(* Logix 5000 project; controller P4 vendor 1 type 14 code 92 rev 20.55; software revision 20.01 *)

TASK MainTask (continuous, watchdog 500 ms) : MainProgram

MODULES
   Local : vendor 1 type 14 code 92 (ICP 0, rev 20.55)
      P4_EN2T_PCN : 1756-EN2T (ICP 1, Ethernet 192.168.1.40, rev 10.1)
         P5 : 1756-EN2T (Ethernet 192.168.1.50, rev 10.1, Output RPI 10 ms)
            P5_CONTROLLER : vendor 1 type 14 code 92 (ICP 0, rev 20.1)
         P3 : 1756-EN2T (Ethernet 192.168.1.30, rev 10.7, Output RPI 10 ms)
            P3_CONTROLLER : vendor 1 type 14 code 92 (ICP 0, rev 20.55)
      P4_EN2TR_RIO : vendor 1 type 12 code 200 (ICP 2, Ethernet 192.168.0.40, rev 10.1)
         RIO4 : 1794-AENTR (Ethernet 192.168.0.42, rev 1.1, Output RPI 20 ms)
            RIO4_DI : 1794-IB32 (Flex 0, rev 1.1, Input RPI 20 ms)
            RIO4_DO : vendor 1 type 7 code 35 (Flex 1, rev 1.1)
            RIO4_AI : 1794-IE12 (Flex 2, rev 1.1, Output RPI 78 ms)
         WRIO4 : vendor 309 type 12 code 1000 (Ethernet 192.168.0.45, rev 3.1, Output RPI 20 ms)
            WRIO3_AI : 1734-IE4C (PointIO 1, rev 3.1, Input RPI 80 ms)
END_MODULES

TYPE AIN_UDT :
STRUCT
   Pv : REAL;
   Heu : REAL;
   Leu : REAL;
   SAHH : REAL;
   SAH : REAL;
   SAL : REAL;
   SALL : REAL;
   AHH : BOOL;
   AH : BOOL;
   AL : BOOL;
   ALL : BOOL;
   Wifi_Enb : BOOL;
   Hty : BOOL;
   Sim : BOOL;
   Sim_PV : REAL;
END_STRUCT
END_TYPE

TYPE AUTOINP_UDT :
STRUCT
   ON : BOOL;
END_STRUCT
END_TYPE

TYPE ControllerLEDStatus :
STRUCT
   Off : BOOL;
   SolidGreen : BOOL;
   FlashingGreen : BOOL;
   SolidYellow : BOOL;
   FlashingYellow : BOOL;
   FlashingRed : BOOL;
   SolidRed : BOOL;
END_STRUCT
END_TYPE

TYPE DOSING_SETPOINT_UDT :
STRUCT
   High_Setpoint : REAL;
   Low_Setpoint : REAL;
END_STRUCT
END_TYPE

TYPE Duty2_UDT :
STRUCT
   Selection : INT;
   Pump_Running : BOOL;
   Selected_Pmp_Not_Avl : BOOL;
   Both_Pmp_Not_Avl : BOOL;
END_STRUCT
END_TYPE

TYPE FaultRecord :
STRUCT
   timelow : DINT;
   timehigh : DINT;
   type : INT;
   code : INT;
   info : DINT[8];
END_STRUCT
END_TYPE

TYPE FIT_UDT :
STRUCT
   Pv : REAL;
   Heu : REAL;
   Leu : REAL;
   SAHH : REAL;
   SAH : REAL;
   SAL : REAL;
   SALL : REAL;
   Totaliser : REAL;
   AHH : BOOL;
   AH : BOOL;
   AL : BOOL;
   ALL : BOOL;
   Sim : BOOL;
   Sim_PV : REAL;
   Wifi_Enb : BOOL;
   Rst_Totaliser : BOOL;
   Hty : BOOL;
END_STRUCT
END_TYPE

TYPE Logix_Status_FP :
STRUCT
   ClearMinorFaults : DINT;
   Sts_MinorFaultEvents : DINT;
   Sts_MinorFaultBits : DINT;
   Sts_Redundant : DINT;
   Set_FaceplateAnimation : DINT;
   Val_ProductCode : DINT;
   MemoryTemp : INT[29];
   Val_raw_data : INT;
   Sts_IO_LED_raw : INT;
   Sts_ProductCode : INT;
   Val_Force_data_raw : INT;
   MemoryRequestData : SINT[12];
   Sts_Force_Installed : BOOL;
   Sts_Force_Enabled : BOOL;
   Sts_Faulted : BOOL;
   Sts_Run : BOOL;
   Sts_Program : BOOL;
   Sts_Minor_fault : BOOL;
   Sts_Major_fault : BOOL;
   Sts_KS_in_run : BOOL;
   Sts_KS_in_program : BOOL;
   Sts_KS_in_remote : BOOL;
   Sts_Changingmodes : BOOL;
   Sts_Test : BOOL;
   Sts_Ladder_Working : BOOL;
   Cmd_ClearFaultRecord : BOOL;
   Set_Controller_Description : STRING;
   UpdateDelayTimer : TIMER;
   Val_MajorFault : FaultRecord;
   Val_MFS : FaultRecord;
   Sts_IO_LED : ControllerLEDStatus;
   Sts_Battery_LED : ControllerLEDStatus;
   MemoryData : Memory_Data;
   TEST : DINT;
END_STRUCT
END_TYPE

TYPE Memory_Data :
STRUCT
   Free_Mem_IO : DINT;
   Free_Mem_DT : DINT;
   Free_Memory : DINT;
   Total_Mem_IO : DINT;
   Total_Mem_DT : DINT;
   Total_Memory : DINT;
   Biggest_IO_Mem_Size_Ava : DINT;
   Biggest_DT_Mem_Size_Ava : DINT;
END_STRUCT
END_TYPE

TYPE MV_UDT :
STRUCT
   Cmd : INT;
   Status : INT;
   Reset : BOOL;
   Auto : BOOL;
   FTO : BOOL;
   FTC : BOOL;
   Avl : BOOL;
END_STRUCT
END_TYPE

TYPE PLANT_AUTO_UDT :
STRUCT
   ON : BOOL;
   OFF : BOOL;
END_STRUCT
END_TYPE

TYPE PLANT_UDT :
STRUCT
   START : BOOL;
   STOP : BOOL;
END_STRUCT
END_TYPE

TYPE PMP_UDT :
STRUCT
   Cmd : INT;
   Status : INT;
   RunMin : REAL;
   Total_RunMin : REAL;
   RunHr : REAL;
   Total_RunHr : REAL;
   Remote : BOOL;
   Auto : BOOL;
   Fault : BOOL;
   Avl : BOOL;
   Permissive : DINT;
   Shutdown : DINT;
   SD : DINT;
   Reset : BOOL;
   Reset_RunHr : BOOL;
   FTR : BOOL;
   FTS : BOOL;
END_STRUCT
END_TYPE

TYPE PRECONDITION_UDT :
STRUCT
   PERMISSIVE1 : BOOL;
   PERMISSIVE2 : BOOL;
   PERMISSIVE3 : BOOL;
   PERMISSIVE4 : BOOL;
   PERMISSIVE5 : BOOL;
   SHUTDOWN1 : BOOL;
   SHUTDOWN2 : BOOL;
   SHUTDOWN3 : BOOL;
   SHUTDOWN4 : BOOL;
   SHUTDOWN5 : BOOL;
END_STRUCT
END_TYPE

TYPE RED_STAT :
STRUCT
   Redundancy_status_of_the_controller : INT;
   Redundancy_state_of_the_partner : INT;
END_STRUCT
END_TYPE

TYPE SWITCH_UDT :
STRUCT
   Alarm : BOOL;
   Delay : DINT;
END_STRUCT
END_TYPE

TYPE UV_UDT :
STRUCT
   Cmd : INT;
   Status : INT;
   RunMin : REAL;
   Total_RunMin : REAL;
   RunHr : REAL;
   Total_RunHr : REAL;
   Remote : BOOL;
   Auto : BOOL;
   Fault : BOOL;
   Avl : BOOL;
   Permissive : DINT;
   Shutdown : DINT;
   SD : DINT;
   Reset : BOOL;
   Reset_RunHr : BOOL;
   FTR : BOOL;
   FTS : BOOL;
END_STRUCT
END_TYPE

TYPE WIFI_UDT :
STRUCT
   PLC_WIFI : BOOL;
   RIO_WIFI : BOOL;
END_STRUCT
END_TYPE

ADD_ON_INSTRUCTION AIN_FBD   (* revision 1.0 *)
VAR_INPUT
   WRIO_Enb : BOOL; {visible}
   Raw_RIO : INT; {visible}
   Raw_WRIO : INT; {visible}
   L_Raw_RIO : INT; {visible}
   H_Raw_RIO : INT; {visible}
   L_Raw_WRIO : INT; {visible}
   H_Raw_WRIO : INT; {visible}
   HEU : INT; {visible}
   LEU : INT; {visible}
END_VAR
VAR_OUTPUT
   Hty : BOOL; {visible}
   Wifi_Enb : BOOL; {access Read Only, visible}
   AHH : BOOL; {visible}
   AH : BOOL; {access Read Only, visible}
   AL : BOOL; {access Read Only, visible}
   ALL : BOOL; {visible}
END_VAR
VAR_INPUT
   SAHH : REAL; {visible}
   SAH : REAL; {visible}
   SAL : REAL; {visible}
   SALL : REAL; {visible}
   Simulation : BOOL; {visible}
   RIO_Hty : BOOL; {visible}
   WRIO_Hty : BOOL; {visible}
END_VAR
VAR_IN_OUT
   Pv : REAL; {required}
   Sim_PV : REAL; {required}
   HMI : AIN_UDT; {required}
END_VAR
VAR
   SCALE : SCALE; {access None}
   ALM : ALARM; {access None}
   _Raw : INT; {access None}
   _L_Raw : INT; {access None}
   _H_Raw : INT; {access None}
   _Inst_Hty : BOOL; {access None}
END_VAR

ROUTINE Logic   (* structured text *)
   (*RIO and Wireless RIO Selection*)
   
   IF WRIO_Enb THEN
   	Wifi_Enb	:= 1;
   	_Raw		:= Raw_WRIO;
   	_H_Raw		:= H_Raw_WRIO;
   	_L_Raw		:= L_Raw_WRIO;
   	_Inst_Hty 	:= WRIO_Hty;
   ELSE
   	Wifi_Enb	:= 0;
   	_Raw		:= Raw_RIO;
   	_H_Raw		:= H_Raw_RIO;
   	_L_Raw		:= L_Raw_RIO;
   	_Inst_Hty 	:= RIO_Hty;
   END_IF;
   
   (*Calculation for PV*)
   IF Simulation THEN
   	Pv	:=Sim_PV;
   ELSE
   	SCALE.In		:=_Raw;
   	SCALE.InRawMax	:=_H_Raw;
   	SCALE.InRawMin	:=_L_Raw;
   	SCALE.InEUMax	:=HEU;
   	SCALE.InEUMin	:=LEU;
   	SCL(SCALE);
   
   	IF SCALE.Out<0 THEN
   		Pv	:= 0.0;
   	ELSE
   		Pv	:=SCALE.Out;
   	END_IF;
   
   	Sim_PV	:=Pv;
   
   END_IF;
   
   (*Alarms*)
   ALM.In			:=Pv;
   ALM.HHLimit		:=SAHH;
   ALM.HLimit		:=SAH;
   ALM.LLimit		:=SAL;
   ALM.LLLimit		:=SALL;
   ALM(ALM);
   
   AHH				:=ALM.HHAlarm;
   AH				:=ALM.HAlarm;
   AL				:=ALM.LAlarm;
   ALL				:=ALM.LLAlarm;
   
   Hty:= _Inst_Hty AND (_Raw > _L_Raw) AND (_Raw < _H_Raw)  ;
   
   
   
   
   
   
END_ROUTINE
END_ADD_ON_INSTRUCTION

ADD_ON_INSTRUCTION Duty2_FBD   (* revision 1.0 *)
VAR_INPUT
   AutoInp : BOOL; {visible}
   Selection : INT; {visible}
END_VAR
VAR_OUTPUT
   Start_Pmp1 : BOOL; {visible}
   Start_Pmp2 : BOOL; {visible}
END_VAR
VAR_IN_OUT
   PMP1 : PMP_UDT; {required}
   PMP2 : PMP_UDT; {required}
   HMI : Duty2_UDT; {required}
END_VAR

ROUTINE Logic   (* structured text *)
   IF PMP1.Status=2 OR PMP2.Status=2 THEN
   	HMI.Pump_Running := 1;
   ELSE
   	HMI.Pump_Running := 0;
   END_IF;
   
   HMI.Both_Pmp_Not_Avl		:= NOT PMP1.Avl AND NOT PMP2.Avl;
   
   IF AutoInp THEN
   	CASE Selection OF
   		(*PUMP 1 *)
   		1:
   			IF PMP1.Avl THEN
   				Start_Pmp1					:=1;
   				Start_Pmp2					:=0;
   				HMI.Selected_Pmp_Not_Avl	:=0;
   			ELSIF NOT PMP1.Avl AND PMP2.Avl THEN
   				Start_Pmp1					:=0;
   				Start_Pmp2					:=1;
   				HMI.Selected_Pmp_Not_Avl	:=1;
   			ELSIF NOT PMP1.Avl AND NOT PMP2.Avl	THEN
   				Start_Pmp1					:=0;
   				Start_Pmp2					:=0;
   			ELSE
   				HMI.Selected_Pmp_Not_Avl	:=0;
   			END_IF;
   
   		(*PUMP 2 *)
   		2:
   			IF PMP2.Avl THEN
   				Start_Pmp1					:=0;
   				Start_Pmp2					:=1;
   				HMI.Selected_Pmp_Not_Avl	:=0;
   			ELSIF NOT PMP2.Avl AND PMP1.Avl THEN
   				Start_Pmp1					:=1;
   				Start_Pmp2					:=0;
   				HMI.Selected_Pmp_Not_Avl	:=1;
   			ELSIF NOT PMP1.Avl AND NOT PMP2.Avl	THEN
   				Start_Pmp1					:=0;
   				Start_Pmp2					:=0;
   			ELSE
   				HMI.Selected_Pmp_Not_Avl	:=0;
   			END_IF;
   	END_CASE;
   ELSE
   	Start_Pmp1					:=0;
   	Start_Pmp2					:=0;
   END_IF;
   
   
END_ROUTINE
END_ADD_ON_INSTRUCTION

ADD_ON_INSTRUCTION FIT_FBD   (* revision 1.0 *)
VAR_INPUT
   WRIO_Enb : BOOL; {visible}
   Raw_RIO : INT; {visible}
   Raw_WRIO : INT; {visible}
   L_Raw_RIO : INT; {visible}
   H_Raw_RIO : INT; {visible}
   L_Raw_WRIO : INT; {visible}
   H_Raw_WRIO : INT; {visible}
   HEU : REAL; {visible}
   LEU : REAL; {visible}
END_VAR
VAR_OUTPUT
   Hty : BOOL; {visible}
   Wifi_Enb : BOOL; {visible}
   AHH : BOOL; {visible}
   AH : BOOL; {access Read Only, visible}
   AL : BOOL; {access Read Only, visible}
   ALL : BOOL; {visible}
END_VAR
VAR_INPUT
   SAHH : REAL; {visible}
   SAH : REAL; {visible}
   SAL : REAL; {visible}
   SALL : REAL; {visible}
   Simulation : BOOL; {visible}
   RIO_Hty : BOOL; {visible}
   WRIO_Hty : BOOL; {visible}
   Totaliser_Enb : BOOL; {visible}
   Rst_Totaliser : BOOL; {visible}
END_VAR
VAR_IN_OUT
   Totaliser : REAL; {required}
   Pv : REAL; {required}
   Sim_Pv : REAL; {required}
   HMI : FIT_UDT; {required}
END_VAR
VAR
   SCALE : SCALE; {access None}
   ALM : ALARM; {access None}
   TON : FBD_TIMER; {access None}
   _SEC_P : BOOL; {access None}
   _Inst_Hty : BOOL; {access None}
   _L_Raw : INT; {access None}
   _H_Raw : INT; {access None}
   _Raw : INT; {access None}
   R_TRIG : FBD_ONESHOT; {access None}
END_VAR

ROUTINE Logic   (* structured text *)
   (*RIO and Wireless RIO Selection*)
   
   IF WRIO_Enb THEN
   	Wifi_Enb	:= 1;
   	_Raw		:= Raw_WRIO;
   	_H_Raw		:= H_Raw_WRIO;
   	_L_Raw		:= L_Raw_WRIO;
   	_Inst_Hty 	:= WRIO_Hty;
   ELSE
   	Wifi_Enb	:= 0;
   	_Raw		:= Raw_RIO;
   	_H_Raw		:= H_Raw_RIO;
   	_L_Raw		:= L_Raw_RIO;
   	_Inst_Hty 	:= RIO_Hty;
   END_IF;
   
   (*Calculation for PV*)
   IF Simulation THEN
   	Pv	:= Sim_Pv   ;
   ELSE
   	SCALE.In		:=_Raw;
   	SCALE.InRawMax	:=_H_Raw;
   	SCALE.InRawMin	:=_L_Raw;
   	SCALE.InEUMax	:=HEU;
   	SCALE.InEUMin	:=LEU;
   	SCL(SCALE);
   	IF SCALE.Out>0 THEN
   		Pv	:=SCALE.Out;
   	ELSIF SCALE.Out<=0 THEN
   		Pv	:=0.0;
   	END_IF;
   
   	Sim_Pv	:=Pv;
   END_IF;
   
   (*Alarms*)
   ALM.In			:=Pv;
   ALM.HHLimit		:=SAHH;
   ALM.HLimit		:=SAH;
   ALM.LLimit		:=SAL;
   ALM.LLLimit		:=SALL;
   ALM(ALM);
   
   AHH				:=ALM.HHAlarm;
   AH				:=ALM.HAlarm;
   AL				:=ALM.LAlarm;
   ALL				:=ALM.LLAlarm;
   
   (*SECOND PULSE*)
   TON.PRE	:=1000;
   TON.TimerEnable	:=1;
   TONR(TON );
   R_TRIG.InputBit :=TON.DN ;
   OSRI( R_TRIG);
   _SEC_P  := R_TRIG.OutputBit;
   TON.Reset := _SEC_P;
   
   IF Totaliser_Enb THEN
   	IF _SEC_P THEN
   		HMI.Totaliser := HMI.Totaliser +  (ABS(Pv) / 3600 );
   	END_IF;
   END_IF;
   
   IF  Rst_Totaliser   THEN
   	HMI.Totaliser	:=0;
   END_IF;
   
   Hty:= _Inst_Hty AND (_Raw > _L_Raw) AND (_Raw < _H_Raw)  ;
   
   
   
   
   
   
END_ROUTINE
END_ADD_ON_INSTRUCTION

ADD_ON_INSTRUCTION MV_FBD   (* revision 1.0 *)
VAR_INPUT
   Auto : BOOL; {visible}
END_VAR
VAR_OUTPUT
   Cmd_Open : BOOL; {visible}
   Cmd_Close : BOOL; {visible}
   FTO : BOOL; {visible}
   FTC : BOOL; {access Read Only, visible}
END_VAR
VAR_INPUT
   AutoInp : BOOL; {visible}
   ZSO : BOOL; {visible}
   Open_TM : DINT; {visible}
   ZSC : BOOL; {visible}
   Close_TM : DINT; {visible}
END_VAR
VAR_IN_OUT
   Cmd : INT; {required}
   HMI : MV_UDT; {required}
END_VAR
VAR
   TON_Open_TM : FBD_TIMER; {access None}
   TON_Close_TM : FBD_TIMER; {access None}
END_VAR

ROUTINE Logic   (* structured text *)
   (*Fail to Close*)
   TON_Close_TM.PRE 			:= 	Close_TM*1000;
   TON_Close_TM.TimerEnable 	:=  Cmd_Close;
   TONR(TON_Close_TM);
   
   (*Fail to Open*)
   TON_Open_TM.PRE 			:= 	Open_TM*1000;
   TON_Open_TM.TimerEnable 	:= 	Cmd_Open;
   TONR(TON_Open_TM);
   
   IF ZSC THEN
   	HMI.Status	:=1;
   ELSIF ZSO THEN
   	HMI.Status	:=2;
   ELSE
   	HMI.Status	:=0;
   END_IF;
   
   HMI.Avl:= Auto AND NOT FTC AND NOT FTO;
   
   IF HMI.Reset THEN
   	(*IF NOT TON_Close_TM.DN AND ZSC THEN*)
   			FTC		:= 0;
   	(*END_IF;*)
   	(*IF NOT TON_Open_TM.DN AND ZSO THEN*)
   			FTO		:= 0;
   	(*END_IF;*)
   END_IF;
   
   IF  NOT Auto THEN
   	CASE HMI.Cmd OF
   		1:	(*CLOSE*)
   			Cmd_Close	:= 1;
   			Cmd_Open	:= 0;
   			IF TON_Close_TM.DN AND (NOT ZSC) THEN
   				FTC		:= 1;
   				FTO		:= 0;
   			END_IF;
   		2:	(*OPEN*)
   			IF FTO OR FTC    THEN
   				HMI.Cmd := 1;
   			END_IF;
   
   			IF NOT FTC AND NOT FTO THEN
   				Cmd_Close	:= 0;
   				Cmd_Open	:= 1;
   			END_IF;
   
   			IF TON_Open_TM.DN AND (NOT ZSO) THEN
   				FTC		:= 0;
   				FTO		:= 1;
   				HMI.Cmd := 1;
   			END_IF;
   	END_CASE;
   ELSE
   	(*Maintain Last status when switching from Auto to Manual*)
   	IF ZSO THEN
   		Cmd	:= 2;
   	END_IF;
   	IF ZSC THEN
   		Cmd	:= 1;
   	END_IF;
   
   	IF  AutoInp AND (NOT FTC AND NOT FTO) THEN
   		Cmd_Close	:= 0;
   		Cmd_Open	:= 1;
   		IF TON_Open_TM.DN AND (NOT ZSO) THEN
   			FTC		:= 0;
   			FTO		:= 1;
   		END_IF;
   	ELSE
   		Cmd_Close	:= 1;
   		Cmd_Open	:= 0;
   		IF TON_Close_TM.DN AND (NOT ZSC) THEN
   			FTC		:= 1;
   			FTO		:= 0;
   		END_IF;
   	END_IF;
   END_IF;
   
   
END_ROUTINE
END_ADD_ON_INSTRUCTION

ADD_ON_INSTRUCTION PMP_FBD   (* revision 1.0 *)
VAR_OUTPUT
   Cmd_Start : BOOL; {visible}
   Avl : BOOL; {visible}
   Fault : BOOL; {visible}
   FT_Stop : BOOL; {visible}
   FT_Start : BOOL; {visible}
   RunHr : REAL; {visible}
   Total_RunHr : REAL; {visible}
   SD : DINT; {access Read Only, visible}
END_VAR
VAR_INPUT
   Auto : BOOL; {visible}
   AutoInp : BOOL; {visible}
   Remote : BOOL; {visible}
   Run : BOOL; {visible}
   Trip : BOOL; {visible}
   Start_TM : DINT; {visible}
   Stop_TM : DINT; {visible}
   Rst : BOOL; {visible}
   Rst_RunHr : BOOL; {visible}
   Permissive : DINT; {visible}
   Shutdown : DINT; {visible}
END_VAR
VAR_IN_OUT
   RunMin : REAL; {required}
   Total_RunMin : REAL; {required}
   Cmd : INT; {required}
   HMI : PMP_UDT; {required}
END_VAR
VAR
   TON_Start_TM : FBD_TIMER; {access None}
   TON_Stop_TM : FBD_TIMER; {access None}
   _Min_P : BOOL; {access None}
   TON_Min : FBD_TIMER; {access None}
   R_TRIG_SEC : FBD_ONESHOT; {access None}
END_VAR

ROUTINE Logic   (* structured text *)
   (*Fail to Start*)
   TON_Start_TM.PRE 			:= 	Start_TM*1000;
   TON_Start_TM.TimerEnable 	:=  Cmd_Start;
   TONR(TON_Start_TM);
   
   (*Fail to Stop*)
   TON_Stop_TM.PRE 			:= 	Stop_TM*1000;
   TON_Stop_TM.TimerEnable 	:=  NOT Cmd_Start;
   TONR(TON_Stop_TM);
   
   IF (NOT Run) THEN
   	HMI.Status	:=1;
   ELSE
   	HMI.Status	:=2;
   END_IF;
   
   IF Fault THEN
   	HMI.Fault:= 1;
   ELSE
   	HMI.Fault:= 0;
   END_IF;
   
   IF HMI.Reset THEN
   	IF NOT TON_Stop_TM.DN THEN
   			FT_Stop		:= 0;
   	END_IF;
   	IF NOT TON_Start_TM.DN THEN
   			FT_Start	:= 0;
   	END_IF;
   
   	SD :=0;
   
   END_IF;
   
   Fault		:=Trip OR SD<>0;
   HMI.Remote	:=Remote;
   Avl:= Auto AND Remote AND NOT Fault AND NOT FT_Start AND NOT FT_Stop AND SD=0 ;
   
   IF Remote THEN
   	IF  NOT Auto THEN
   		CASE HMI.Cmd OF
   			1:	(*Stop*)
   				Cmd_Start	:=0;
   				IF TON_Stop_TM.DN AND Run THEN
   					FT_Start	:= 0;
   					FT_Stop		:= 1;
   				END_IF;
   			2:	(*OPEN*)
   				IF NOT Fault AND NOT FT_Start AND NOT FT_Stop AND (Permissive=-1) AND HMI.SD=0 THEN
   					Cmd_Start	:= 1;
   				ELSIF Cmd_Start AND (HMI.SD<>0) OR Fault THEN
   					SD				:= HMI.SD;
   					Cmd_Start		:= 0;
   					HMI.Cmd 		:= 1;
   				ELSIF (Permissive<>-1) THEN
   					HMI.Cmd 		:= 1;
   				END_IF;
   
   				IF TON_Start_TM.DN AND NOT Run THEN
   					FT_Start	:= 1;
   					FT_Stop		:= 0;
   					Cmd_Start	:= 0;
   					HMI.Cmd 	:= 1;
   				END_IF;
   		END_CASE;
   	ELSE
   		IF Run THEN
   			Cmd	:= 2;
   		END_IF;
   		IF (NOT Run) OR Fault OR FT_Start OR FT_Stop THEN
   			Cmd	:= 1;
   		END_IF;
   
   		IF  AutoInp  THEN
   			IF NOT Fault AND NOT FT_Start AND NOT FT_Stop AND (Permissive=-1) AND HMI.SD=0  THEN
   				Cmd_Start	:=1;
   			ELSIF Cmd_Start OR (HMI.SD<>0) OR Fault THEN
   				SD			:= HMI.SD;
   				Cmd_Start	:=0;
   			END_IF;
   
   			IF TON_Start_TM.DN AND NOT Run THEN
   				FT_Start	:= 1;
   				FT_Stop		:= 0;
   				Cmd_Start	:= 0;
   				HMI.Cmd 	:= 1;
   			END_IF;
   		ELSE
   			Cmd_Start	:=0;
   			IF TON_Stop_TM.DN AND Run THEN
   				FT_Start	:= 0;
   				FT_Stop		:= 1;
   
   			END_IF;
   		END_IF;
   	END_IF;
   
   ELSE (*Local*)
   	Cmd_Start	:=0;
   	Cmd	:= 1;
   
   	FT_Start	:= 0;
   	FT_Stop		:= 0;
   
   
   
   
   	(*	IF Run THEN
   			Cmd	:= 2;
   		END_IF;
   		IF (NOT Run) OR Fault OR FT_Start OR FT_Stop THEN
   			Cmd	:= 1;
   		END_IF;
   		*)
   END_IF;
   
   (*1 MIN PULSE*)
   TON_Min.PRE	:=60000;
   TON_Min.TimerEnable	:=1;
   TONR(TON_Min );
   R_TRIG_SEC.InputBit :=TON_Min.DN ;
   OSRI( R_TRIG_SEC);
   _Min_P  := R_TRIG_SEC.OutputBit;
   TON_Min.Reset 	:= _Min_P;
   
   IF Run THEN
   	IF _Min_P THEN
   		RunMin 			:=RunMin + 1.0;
   		Total_RunMin	:=Total_RunMin + 1.0;
   	END_IF;
   END_IF;
   
   RunHr 				:=RunMin/60.0;
   Total_RunHr			:=Total_RunMin/60.0;
   
   IF  Rst_RunHr THEN
   	RunMin	:=0;
   END_IF;
   
   
   
END_ROUTINE
END_ADD_ON_INSTRUCTION

ADD_ON_INSTRUCTION SWITCH_FBD   (* revision 1.0 *)
VAR_INPUT
   Alarm : BOOL; {visible}
   Delay : DINT; {required}
END_VAR
VAR_OUTPUT
   Status : BOOL; {access None, required}
END_VAR
VAR_IN_OUT
   HMI : SWITCH_UDT; {required}
END_VAR
VAR
   TON_Delay_Sec : FBD_TIMER; {access None}
END_VAR

ROUTINE Logic   (* structured text *)
   (*Delay for Alarm*)
   TON_Delay_Sec.PRE 			:= 	Delay*1000;
   TON_Delay_Sec.TimerEnable 	:=  Alarm;
   TONR(TON_Delay_Sec);
   
   Status := TON_Delay_Sec.DN ;
END_ROUTINE
END_ADD_ON_INSTRUCTION

ADD_ON_INSTRUCTION UV_FBD   (* revision 1.0 *)
VAR_OUTPUT
   Cmd_Start : BOOL; {visible}
   Avl : BOOL; {visible}
   Fault : BOOL; {visible}
   FT_Stop : BOOL; {visible}
   FT_Start : BOOL; {visible}
   RunHr : REAL; {visible}
   Total_RunHr : REAL; {visible}
   SD : DINT; {visible}
END_VAR
VAR_INPUT
   Auto : BOOL; {visible}
   AutoInp : BOOL; {visible}
   Remote : BOOL; {visible}
   Run : BOOL; {visible}
   Trip : BOOL; {visible}
   Start_TM : DINT; {visible}
   Stop_TM : DINT; {visible}
   Rst : BOOL; {visible}
   Rst_RunHr : BOOL; {visible}
   Permissive : DINT; {visible}
   Shutdown : DINT; {visible}
END_VAR
VAR_IN_OUT
   RunMin : REAL; {required}
   Total_RunMin : REAL; {required}
   Cmd : INT; {required}
   HMI : UV_UDT; {required}
END_VAR
VAR
   TON_Start_TM : FBD_TIMER; {access None}
   TON_Stop_TM : FBD_TIMER; {access None}
   _Min_P : BOOL; {access None}
   TON_Min : FBD_TIMER; {access None}
   R_TRIG_SEC : FBD_ONESHOT; {access None}
END_VAR

ROUTINE Logic   (* structured text *)
   (*Fail to Start*)
   TON_Start_TM.PRE 			:= 	Start_TM*1000;
   TON_Start_TM.TimerEnable 	:=  Cmd_Start;
   TONR(TON_Start_TM);
   
   (*Fail to Stop*)
   TON_Stop_TM.PRE 			:= 	Stop_TM*1000;
   TON_Stop_TM.TimerEnable 	:=  NOT Cmd_Start;
   TONR(TON_Stop_TM);
   
   IF (NOT Run) THEN
   	HMI.Status	:=1;
   ELSE
   	HMI.Status	:=2;
   END_IF;
   
   IF Fault THEN
   	HMI.Fault:= 1;
   ELSE
   	HMI.Fault:= 0;
   END_IF;
   
   IF HMI.Reset THEN
   	IF NOT TON_Stop_TM.DN THEN
   			FT_Stop		:= 0;
   	END_IF;
   	IF NOT TON_Start_TM.DN THEN
   			FT_Start	:= 0;
   	END_IF;
   
   	SD :=0;
   
   END_IF;
   
   Fault		:=Trip;
   HMI.Remote	:=Remote;
   Avl:= Auto AND Remote AND NOT Fault AND NOT FT_Start AND NOT FT_Stop AND SD=0 ;
   
   IF Remote THEN
   	IF  NOT Auto THEN
   		CASE HMI.Cmd OF
   			1:	(*Stop*)
   				Cmd_Start	:=0;
   				IF TON_Stop_TM.DN AND Run THEN
   					FT_Start	:= 0;
   					FT_Stop		:= 1;
   				END_IF;
   			2:	(*OPEN*)
   				IF NOT Fault AND NOT FT_Start AND NOT FT_Stop AND (Permissive=-1) AND HMI.SD=0 THEN
   					Cmd_Start	:= 1;
   				ELSIF Cmd_Start AND (HMI.SD<>0) OR Fault THEN
   					SD				:= HMI.SD;
   					Cmd_Start		:= 0;
   					HMI.Cmd 		:= 1;
   				END_IF;
   
   				IF TON_Start_TM.DN AND NOT Run THEN
   					FT_Start	:= 1;
   					FT_Stop		:= 0;
   					Cmd_Start	:= 0;
   					HMI.Cmd 	:= 1;
   				END_IF;
   		END_CASE;
   	ELSE
   		IF Run THEN
   			Cmd	:= 2;
   		END_IF;
   		IF (NOT Run) OR Fault OR FT_Start OR FT_Stop THEN
   			Cmd	:= 1;
   		END_IF;
   
   		IF  AutoInp  THEN
   			IF NOT Fault AND NOT FT_Start AND NOT FT_Stop AND (Permissive=-1) AND HMI.SD=0  THEN
   				Cmd_Start	:=1;
   			ELSIF Cmd_Start OR (HMI.SD<>0) OR Fault THEN
   				SD			:= HMI.SD;
   				Cmd_Start	:=0;
   			END_IF;
   
   			IF TON_Start_TM.DN AND NOT Run THEN
   				FT_Start	:= 1;
   				FT_Stop		:= 0;
   				Cmd_Start	:= 0;
   				HMI.Cmd 	:= 1;
   			END_IF;
   		ELSE
   			Cmd_Start	:=0;
   			IF TON_Stop_TM.DN AND Run THEN
   				FT_Start	:= 0;
   				FT_Stop		:= 1;
   
   			END_IF;
   		END_IF;
   	END_IF;
   
   ELSE (*Local*)
   	Cmd_Start	:=0;
   	Cmd	:= 1;
   
   	FT_Start	:= 0;
   	FT_Stop		:= 0;
   
   
   
   
   	(*	IF Run THEN
   			Cmd	:= 2;
   		END_IF;
   		IF (NOT Run) OR Fault OR FT_Start OR FT_Stop THEN
   			Cmd	:= 1;
   		END_IF;
   		*)
   END_IF;
   
   (*1 MIN PULSE*)
   TON_Min.PRE	:=60000;
   TON_Min.TimerEnable	:=1;
   TONR(TON_Min );
   R_TRIG_SEC.InputBit :=TON_Min.DN ;
   OSRI( R_TRIG_SEC);
   _Min_P  := R_TRIG_SEC.OutputBit;
   TON_Min.Reset 	:= _Min_P;
   
   IF Run THEN
   	IF _Min_P THEN
   		RunMin 			:=RunMin + 1.0;
   		Total_RunMin	:=Total_RunMin + 1.0;
   	END_IF;
   END_IF;
   
   RunHr 				:=RunMin/60.0;
   Total_RunHr			:=Total_RunMin/60.0;
   
   IF  Rst_RunHr THEN
   	RunMin	:=0;
   END_IF;
   
   
   
END_ROUTINE
END_ADD_ON_INSTRUCTION

VAR_GLOBAL   (* controller tags *)
   _FIT401_Tot_Enb : BOOL;
   _P401_AutoInp : BOOL;
   _P402_AutoInp : BOOL;
   _P403_AutoInp : BOOL;
   _P404_AutoInp : BOOL;
   _P_NAHSO3_ORP_DUTY_AutoInp : BOOL;
   _P_NAHSO3_ORP_DUTY_SR : DOMINANT_SET := (Reset := 1, OutNot := 1);
   _P_RO_FEED_DUTY_AutoInp : BOOL;
   _P_RO_FEED_DUTY_SR : DOMINANT_SET := (Set := 1, Out := 1);
   _P_UF_FEED_DUTY_AutoInp : BOOL := 1;
   _UV401_AutoInp : BOOL;
   _UV_SR : DOMINANT_SET := (Set := 1, Out := 1);
   AI_AIT_401_HRDNSS : INT := 35;
   AI_AIT_401_HRDNSS_HTY : BOOL := 1;
   AI_AIT_402_ORP : INT := 9619;
   AI_AIT_402_ORP_HTY : BOOL := 1;
   AI_FIT_401_FLOW : INT := -7;
   AI_FIT_401_FLOW_HTY : BOOL := 1;
   AI_LIT_401_LEVEL : INT := 20593;
   AI_LIT_401_LEVEL_HTY : BOOL := 1;
   AI_RIO4_SPARE_03 : INT := 9619;
   AI_RIO4_SPARE_03_HTY : BOOL := 1;
   AI_RIO4_SPARE_04 : INT := -7703;
   AI_RIO4_SPARE_04_HTY : BOOL := 1;
   AI_RIO4_SPARE_05 : INT := -7703;
   AI_RIO4_SPARE_05_HTY : BOOL := 1;
   AI_RIO4_SPARE_06 : INT := -7698;
   AI_RIO4_SPARE_06_HTY : BOOL := 1;
   AI_RIO4_SPARE_07 : INT := -7702;
   AI_RIO4_SPARE_07_HTY : BOOL := 1;
   AI_RIO4_SPARE_08 : INT := -7699;
   AI_RIO4_SPARE_08_HTY : BOOL := 1;
   AI_RIO4_SPARE_09 : INT := -7702;
   AI_RIO4_SPARE_09_HTY : BOOL := 1;
   AI_RIO4_SPARE_10 : INT := -7701;
   AI_RIO4_SPARE_10_HTY : BOOL := 1;
   AI_RIO4_SPARE_11 : INT := -7703;
   AI_RIO4_SPARE_11_HTY : BOOL := 1;
   AIT401_FB : AIN_FBD := (Raw_RIO := 35, Raw_WRIO := 3261, H_Raw_RIO := 31208, L_Raw_WRIO := 3277, H_Raw_WRIO := 16383, HEU := 150, Hty := 1, AL := 1, ALL := 1, SAHH := 100.0, SAH := 80.0, SAL := 20.0, SALL := 10.0, RIO_Hty := 1, WRIO_Hty := 1);
   AIT401_FB_01 : AIN_FBD;
   AIT402_FB : AIN_FBD := (Raw_RIO := 9619, Raw_WRIO := 8246, H_Raw_RIO := 31208, L_Raw_WRIO := 3277, H_Raw_WRIO := 16383, HEU := 800, Hty := 1, AL := 1, SAHH := 800.0, SAH := 275.0, SAL := 250.0, SALL := 200.0, RIO_Hty := 1);
   DI_DPSH_301_HIGH : BOOL;
   DI_LS_401_LOW : BOOL := 1;
   DI_P_401_AUTO : BOOL := 1;
   DI_P_401_FAULT : BOOL;
   DI_P_401_RUN : BOOL;
   DI_P_402_AUTO : BOOL := 1;
   DI_P_402_FAULT : BOOL;
   DI_P_402_RUN : BOOL;
   DI_P_403_AUTO : BOOL := 1;
   DI_P_403_FAULT : BOOL;
   DI_P_403_RUN : BOOL;
   DI_P_404_AUTO : BOOL := 1;
   DI_P_404_FAULT : BOOL;
   DI_P_404_RUN : BOOL;
   DI_RIO4_SPARE_10 : BOOL;
   DI_RIO4_SPARE_11 : BOOL;
   DI_RIO4_SPARE_12 : BOOL;
   DI_RIO4_SPARE_13 : BOOL;
   DI_RIO4_SPARE_14 : BOOL;
   DI_RIO4_SPARE_15 : BOOL;
   DI_RIO4_SPARE_16 : BOOL;
   DI_RIO4_SPARE_17 : BOOL;
   DI_RIO4_SPARE_18 : BOOL;
   DI_RIO4_SPARE_19 : BOOL;
   DI_RIO4_SPARE_20 : BOOL;
   DI_RIO4_SPARE_21 : BOOL;
   DI_RIO4_SPARE_22 : BOOL;
   DI_RIO4_SPARE_23 : BOOL;
   DI_RIO4_SPARE_24 : BOOL;
   DI_RIO4_SPARE_25 : BOOL;
   DI_RIO4_SPARE_26 : BOOL;
   DI_RIO4_SPARE_27 : BOOL;
   DI_RIO4_SPARE_28 : BOOL;
   DI_RIO4_SPARE_29 : BOOL;
   DI_RIO4_SPARE_30 : BOOL;
   DI_RIO4_SPARE_31 : BOOL;
   DI_UV_401_AUTO : BOOL := 1;
   DI_UV_401_FAULT : BOOL;
   DI_UV_401_RUN : BOOL;
   DI_UV_402_FAULT : BOOL;
   DI_UV_402_RUN : BOOL;
   DI_WIFI_PLC_4 : BOOL;
   DI_WIFI_RIO_4 : BOOL;
   DO_P_401_START : BOOL;
   DO_P_402_START : BOOL;
   DO_P_403_START : BOOL;
   DO_P_404_START : BOOL;
   DO_RIO4_SPARE_04 : BOOL;
   DO_RIO4_SPARE_05 : BOOL;
   DO_RIO4_SPARE_06 : BOOL;
   DO_RIO4_SPARE_07 : BOOL;
   DO_RIO4_SPARE_08 : BOOL;
   DO_RIO4_SPARE_09 : BOOL;
   DO_RIO4_SPARE_10 : BOOL;
   DO_RIO4_SPARE_11 : BOOL;
   DO_RIO4_SPARE_12 : BOOL;
   DO_RIO4_SPARE_13 : BOOL;
   DO_RIO4_SPARE_14 : BOOL;
   DO_RIO4_SPARE_15 : BOOL;
   DO_UV_401_START : BOOL;
   FIT401_FB : FIT_FBD := (Raw_RIO := -7, Raw_WRIO := 3264, L_Raw_RIO := -5, H_Raw_RIO := 31208, L_Raw_WRIO := 3277, H_Raw_WRIO := 16383, HEU := 4.0, AL := 1, ALL := 1, SAHH := 3.0, SAH := 2.0, SAL := 1.0, SALL := 0.5, RIO_Hty := 1, WRIO_Hty := 1);
   HMI_AIT401 : AIN_UDT := (Pv := 0.1682261, SAHH := 100.0, SAH := 80.0, SAL := 20.0, SALL := 10.0, AL := 1, ALL := 1, Hty := 1, Sim_PV := 0.1682261);
   HMI_AIT402 : AIN_UDT := (Pv := 246.5778, SAHH := 800.0, SAH := 275.0, SAL := 250.0, SALL := 200.0, AL := 1, Hty := 1, Sim_PV := 246.5778);
   HMI_FIT401 : FIT_UDT := (SAHH := 3.0, SAH := 2.0, SAL := 1.0, SALL := 0.5, Totaliser := 55.34227, AL := 1, ALL := 1);
   HMI_LIT401 : AIN_UDT := (Pv := 791.83545, SAHH := 1200.0, SAH := 800.0, SAL := 800.0, SALL := 250.0, AL := 1, Hty := 1, Sim_PV := 791.83545);
   HMI_LS401 : SWITCH_UDT;
   HMI_MV302 : MV_UDT := (Cmd := 1, Status := 1, Reset := 1, Auto := 1, Avl := 1);
   HMI_MV501 : MV_UDT := (Cmd := 1, Status := 1, Reset := 1, Auto := 1, Avl := 1);
   HMI_MV502 : MV_UDT := (Cmd := 1, Status := 1, Reset := 1, Auto := 1, Avl := 1);
   HMI_MV503 : MV_UDT := (Cmd := 1, Status := 1, Reset := 1, Auto := 1, Avl := 1);
   HMI_MV504 : MV_UDT := (Cmd := 1, Status := 1, Reset := 1, Auto := 1, Avl := 1);
   HMI_NAHSO3_ORP_DOSING : DOSING_SETPOINT_UDT;
   HMI_P301 : PMP_UDT := (Cmd := 1, Status := 1, RunMin := 2002.0, Total_RunMin := 2002.0, RunHr := 33.366665, Total_RunHr := 33.366665, Remote := 1, Auto := 1, Avl := 1, Permissive := -3, Reset := 1);
   HMI_P301_MSG : PRECONDITION_UDT := (PERMISSIVE1 := 1);
   HMI_P401 : PMP_UDT := (Cmd := 1, Status := 1, RunMin := 2002.0, Total_RunMin := 2002.0, RunHr := 33.366665, Total_RunHr := 33.366665, Remote := 1, Auto := 1, Avl := 1, Permissive := -3, Reset := 1);
   HMI_P401_MSG : PRECONDITION_UDT := (PERMISSIVE1 := 1);
   HMI_P402 : PMP_UDT := (Cmd := 1, Status := 1, RunMin := 748.0, Total_RunMin := 748.0, RunHr := 12.466666, Total_RunHr := 12.466666, Remote := 1, Auto := 1, Avl := 1, Permissive := -3, Reset := 1);
   HMI_P402_MSG : PRECONDITION_UDT := (PERMISSIVE1 := 1);
   HMI_P403 : PMP_UDT := (Cmd := 1, Status := 1, RunMin := 796.0, Total_RunMin := 796.0, RunHr := 13.266666, Total_RunHr := 13.266666, Remote := 1, Auto := 1, Avl := 1, Permissive := -3, Reset := 1);
   HMI_P403_MSG : PRECONDITION_UDT := (PERMISSIVE1 := 1);
   HMI_P404 : PMP_UDT := (Cmd := 1, Status := 1, RunMin := 2.0, Total_RunMin := 2.0, RunHr := 0.033333335, Total_RunHr := 0.033333335, Remote := 1, Auto := 1, Avl := 1, Permissive := -3, Reset := 1);
   HMI_P404_MSG : PRECONDITION_UDT := (PERMISSIVE1 := 1);
   HMI_P4_PERMISSIVE : AUTOINP_UDT := (ON := 1);
   HMI_P4_STATE : INT := 1;
   HMI_P_NAHSO3_ORP_DUTY : Duty2_UDT := (Selection := 1);
   HMI_P_RO_FEED_DUTY : Duty2_UDT := (Selection := 1);
   HMI_P_UF_FEED_DUTY : Duty2_UDT;
   HMI_PLANT : PLANT_UDT;
   HMI_PLANT_AUTO : PLANT_AUTO_UDT;
   HMI_PLANT_PERMISSIVE : BOOL := 1;
   HMI_PLANT_RESET : PLANT_AUTO_UDT;
   HMI_RO_HPP_SD : AUTOINP_UDT;
   HMI_START_PLANT : BOOL;
   HMI_UV401 : UV_UDT := (Cmd := 1, Status := 1, RunMin := 2747.0, Total_RunMin := 2747.0, RunHr := 45.783333, Total_RunHr := 45.783333, Remote := 1, Auto := 1, Avl := 1, Permissive := -4, Reset := 1);
   HMI_UV401_MSG : PRECONDITION_UDT := (PERMISSIVE1 := 1);
   HMI_UV404_MSG : PRECONDITION_UDT;
   HMI_WIFI : WIFI_UDT;
   LIT401_FB : AIN_FBD := (Raw_RIO := 20597, Raw_WRIO := 14965, H_Raw_RIO := 31208, L_Raw_WRIO := 3277, H_Raw_WRIO := 16383, HEU := 1200, Hty := 1, AL := 1, SAHH := 1200.0, SAH := 800.0, SAL := 800.0, SALL := 250.0, RIO_Hty := 1, WRIO_Hty := 1);
   LIT401_FB_01 : AIN_FBD;
   Logix_Status : Logix_Status_FP := (Set_FaceplateAnimation := 90, Val_ProductCode := 92, MemoryTemp[0] := 5, MemoryTemp[1] := 1, MemoryTemp[3] := 31408, MemoryTemp[4] := 3, MemoryTemp[5] := 15230, MemoryTemp[6] := 7, MemoryTemp[9] := 2, MemoryTemp[11] := -4608, MemoryTemp[12] := 3, MemoryTemp[14] := 8, MemoryTemp[17] := 5, MemoryTemp[21] := 6, MemoryTemp[23] := 30650, MemoryTemp[24] := 3, MemoryTemp[25] := 7, MemoryTemp[27] := 8988, MemoryTemp[28] := 7, Val_raw_data := 12640, Sts_IO_LED_raw := 2, Sts_ProductCode := 92, MemoryRequestData[0] := 5, MemoryRequestData[2] := 1, MemoryRequestData[4] := 2, MemoryRequestData[6] := 5, MemoryRequestData[8] := 6, MemoryRequestData[10] := 7, Sts_Run := 1, Sts_KS_in_remote := 1, Sts_Ladder_Working := 1, Set_Controller_Description := 'P4: De-Chlorination System', UpdateDelayTimer.PRE := 1000, UpdateDelayTimer.ACC := 43, UpdateDelayTimer.EN := 1, UpdateDelayTimer.TT := 1, Val_MFS.timelow := 71751885, Val_MFS.timehigh := 206334, Val_MFS.type := 3, Val_MFS.code := 20, Val_MFS.info[1] := 1, Sts_IO_LED.FlashingGreen := 1, Sts_Battery_LED.Off := 1, MemoryData.Free_Mem_IO := 912064, MemoryData.Free_Mem_DT := 1895928, MemoryData.Total_Mem_IO := 1030144, MemoryData.Total_Mem_DT := 2097152, MemoryData.Biggest_IO_Mem_Size_Ava := 909032, MemoryData.Biggest_DT_Mem_Size_Ava := 1870960);
   LS401_FB : SWITCH_FBD;
   Memory_Message : MESSAGE;
        MessageParameters(ServiceCode := 16#0003, LocalElement := Logix_Status.MemoryRequestData[0], DestinationTag := Logix_Status.MemoryTemp[0], ...)
   P3_MV302_MSG : MESSAGE;
        MessageParameters(ServiceCode := 16#004c, LocalElement := HMI_MV302, ...)
   P3_P301_MSG : MESSAGE;
        MessageParameters(ServiceCode := 16#004c, LocalElement := HMI_P301, ...)
   P401_FB : PMP_FBD := (Avl := 1, RunHr := 33.366665, Total_RunHr := 33.366665, Auto := 1, Remote := 1, Start_TM := 3, Stop_TM := 3, Rst := 1, Permissive := -3);
   P402_FB : PMP_FBD := (Avl := 1, RunHr := 12.466666, Total_RunHr := 12.466666, Auto := 1, Remote := 1, Start_TM := 3, Stop_TM := 3, Rst := 1, Permissive := -3);
   P403_FB : PMP_FBD := (Avl := 1, RunHr := 13.266666, Total_RunHr := 13.266666, Auto := 1, Remote := 1, Start_TM := 3, Stop_TM := 3, Rst := 1, Permissive := -3);
   P404_FB : PMP_FBD := (Avl := 1, RunHr := 0.033333335, Total_RunHr := 0.033333335, Auto := 1, Remote := 1, Start_TM := 3, Stop_TM := 3, Rst := 1, Permissive := -3);
   P5_MV501_MSG : MESSAGE;
        MessageParameters(ServiceCode := 16#004c, LocalElement := HMI_MV501, ...)
   P5_MV502_MSG : MESSAGE;
        MessageParameters(ServiceCode := 16#004c, LocalElement := HMI_MV502, ...)
   P5_MV503_MSG : MESSAGE;
        MessageParameters(ServiceCode := 16#004c, LocalElement := HMI_MV503, ...)
   P5_MV504_MSG : MESSAGE;
        MessageParameters(ServiceCode := 16#004c, LocalElement := HMI_MV504, ...)
   P_NAHSO3_ORP_DUTY_FB : Duty2_FBD := (Selection := 1);
   P_RO_FEED_DUTY_FB : Duty2_FBD := (Selection := 1);
   R_TRIG : FBD_ONESHOT;
   REDUNDANT_STATUS : RED_STAT := (Redundancy_status_of_the_controller := 2, Redundancy_state_of_the_partner := 8);
   TON : FBD_TIMER := (TimerEnable := 1, PRE := 1000, ACC := 475, EN := 1, TT := 1);
   TON_FIT401_P1_TM : FBD_TIMER := (PRE := 6000);
   TON_FIT401_P2_TM : FBD_TIMER := (PRE := 6000);
   TON_FIT401_TM : FBD_TIMER := (PRE := 6000);
   UV401_FB : UV_FBD := (Avl := 1, RunHr := 45.783333, Total_RunHr := 45.783333, Auto := 1, Remote := 1, Start_TM := 3, Stop_TM := 3, Rst := 1, Permissive := -4);
   W_AI_AIT_401_HRDNSS : INT := 3261;
   W_AI_AIT_401_HRDNSS_HTY : BOOL := 1;
   W_AI_AIT_402_ORP : INT := 8246;
   W_AI_AIT_402_ORP_HTY : BOOL;
   W_AI_FIT_401_FLOW : INT := 3264;
   W_AI_FIT_401_FLOW_HTY : BOOL := 1;
   W_AI_LIT_301_LEVEL : INT;
   W_AI_LIT_301_LEVEL_HTY : BOOL;
   W_AI_LIT_401_LEVEL : INT := 14965;
   W_AI_LIT_401_LEVEL_HTY : BOOL := 1;
   W_AI_RIO4_SPARE_03_HTY : BOOL := 1;
END_VAR

PROGRAM MainProgram   (* main routine MainRoutine *)
VAR
   _MIN_P : BOOL;
   _SEC_P : BOOL;
   ATTACK : BOOL;
   Duty2_FBD_01 : Duty2_FBD;
   PMP_FBD_01 : PMP_FBD;
   PMP_FBD_02 : PMP_FBD;
   SEC_TEST : DINT;
   UV_FBD_01 : UV_FBD;
END_VAR

ROUTINE Dosing   (* function block diagram *)
   SHEET 1
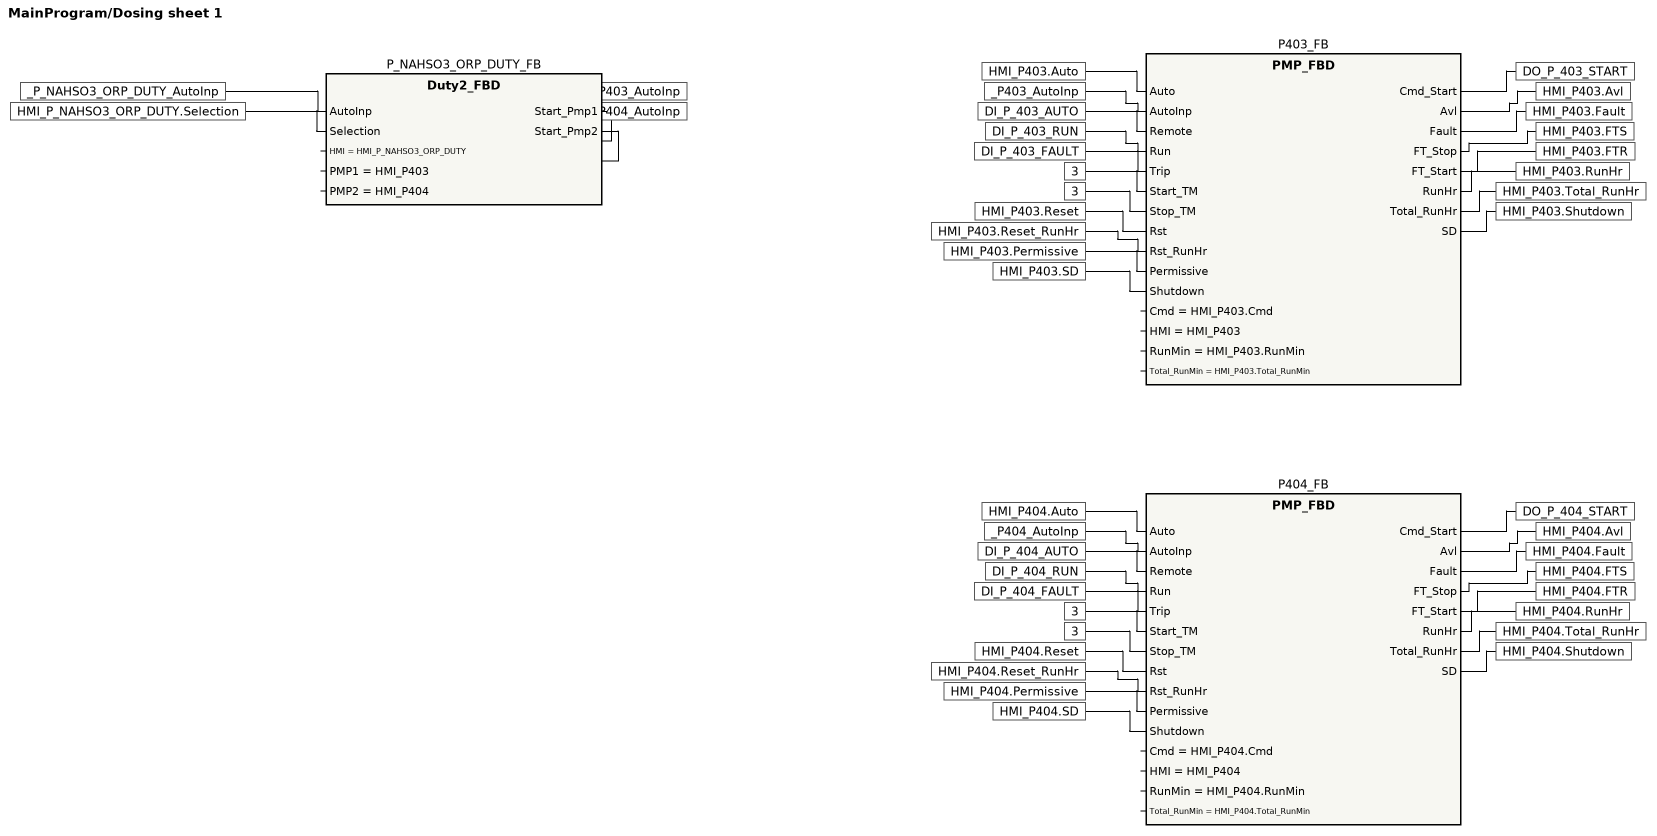
   P_NAHSO3_ORP_DUTY_FB : Duty2_FBD(AutoInp := _P_NAHSO3_ORP_DUTY_AutoInp, Selection := HMI_P_NAHSO3_ORP_DUTY.Selection, HMI := HMI_P_NAHSO3_ORP_DUTY, PMP1 := HMI_P403, PMP2 := HMI_P404);
   _P403_AutoInp := P_NAHSO3_ORP_DUTY_FB.Start_Pmp1;
   _P404_AutoInp := P_NAHSO3_ORP_DUTY_FB.Start_Pmp2;
   P403_FB : PMP_FBD(Auto := HMI_P403.Auto, AutoInp := _P403_AutoInp, Remote := DI_P_403_AUTO, Run := DI_P_403_RUN, Trip := DI_P_403_FAULT, Start_TM := 3, Stop_TM := 3, Rst := HMI_P403.Reset, Rst_RunHr := HMI_P403.Reset_RunHr, Permissive := HMI_P403.Permissive, Shutdown := HMI_P403.SD, Cmd := HMI_P403.Cmd, HMI := HMI_P403, RunMin := HMI_P403.RunMin, Total_RunMin := HMI_P403.Total_RunMin);
   P404_FB : PMP_FBD(Auto := HMI_P404.Auto, AutoInp := _P404_AutoInp, Remote := DI_P_404_AUTO, Run := DI_P_404_RUN, Trip := DI_P_404_FAULT, Start_TM := 3, Stop_TM := 3, Rst := HMI_P404.Reset, Rst_RunHr := HMI_P404.Reset_RunHr, Permissive := HMI_P404.Permissive, Shutdown := HMI_P404.SD, Cmd := HMI_P404.Cmd, HMI := HMI_P404, RunMin := HMI_P404.RunMin, Total_RunMin := HMI_P404.Total_RunMin);
   HMI_P403.Total_RunHr := P403_FB.Total_RunHr;
   HMI_P403.Shutdown := P403_FB.SD;
   HMI_P404.Total_RunHr := P404_FB.Total_RunHr;
   HMI_P404.Shutdown := P404_FB.SD;
   DO_P_403_START := P403_FB.Cmd_Start;
   HMI_P403.RunHr := P403_FB.RunHr;
   DO_P_404_START := P404_FB.Cmd_Start;
   HMI_P404.RunHr := P404_FB.RunHr;
   HMI_P403.Fault := P403_FB.Fault;
   HMI_P404.Fault := P404_FB.Fault;
   HMI_P403.Avl := P403_FB.Avl;
   HMI_P403.FTS := P403_FB.FT_Stop;
   HMI_P403.FTR := P403_FB.FT_Start;
   HMI_P404.Avl := P404_FB.Avl;
   HMI_P404.FTS := P404_FB.FT_Stop;
   HMI_P404.FTR := P404_FB.FT_Start;
END_ROUTINE

ROUTINE IO   (* structured text *)
   (*DIGITAL INPUTS*)
   DI_WIFI_PLC_4	:=RIO4:0:I.Data.0;
   DI_WIFI_RIO_4	:=RIO4:0:I.Data.1;
   DI_P_401_AUTO	:=RIO4:0:I.Data.2;
   DI_P_401_RUN	:=RIO4:0:I.Data.3;
   DI_P_401_FAULT	:=RIO4:0:I.Data.4;
   DI_P_402_AUTO	:=RIO4:0:I.Data.5;
   DI_P_402_RUN	:=RIO4:0:I.Data.6;
   DI_P_402_FAULT	:=RIO4:0:I.Data.7;
   DI_P_403_AUTO	:=RIO4:0:I.Data.8;
   DI_P_403_RUN	:=RIO4:0:I.Data.9;
   DI_P_403_FAULT	:=RIO4:0:I.Data.10;
   DI_P_404_AUTO	:=RIO4:0:I.Data.11;
   DI_P_404_RUN	:=RIO4:0:I.Data.12;
   DI_P_404_FAULT	:=RIO4:0:I.Data.13;
   DI_UV_401_AUTO	:=RIO4:0:I.Data.14;
   DI_UV_401_RUN	:=RIO4:0:I.Data.15;
   DI_UV_401_FAULT	:=RIO4:0:I.Data.16;
   DI_LS_401_LOW	:=RIO4:0:I.Data.17;
   DI_RIO4_SPARE_18:=RIO4:0:I.Data.18;
   DI_RIO4_SPARE_19:=RIO4:0:I.Data.19;
   DI_RIO4_SPARE_20:=RIO4:0:I.Data.20;
   DI_RIO4_SPARE_21:=RIO4:0:I.Data.21;
   DI_RIO4_SPARE_22:=RIO4:0:I.Data.22;
   DI_RIO4_SPARE_23:=RIO4:0:I.Data.23;
   DI_RIO4_SPARE_24:=RIO4:0:I.Data.24;
   DI_RIO4_SPARE_25:=RIO4:0:I.Data.25;
   DI_RIO4_SPARE_26:=RIO4:0:I.Data.26;
   DI_RIO4_SPARE_27:=RIO4:0:I.Data.27;
   DI_RIO4_SPARE_28:=RIO4:0:I.Data.28;
   DI_RIO4_SPARE_29:=RIO4:0:I.Data.29;
   DI_RIO4_SPARE_30:=RIO4:0:I.Data.30;
   DI_RIO4_SPARE_31:=RIO4:0:I.Data.31;
   
   (*DIGITAL OUTPUTS*)
   RIO4:1:O.0	:=DO_P_401_START;
   RIO4:1:O.1	:=DO_P_402_START;
   RIO4:1:O.2	:=DO_P_403_START;
   RIO4:1:O.3	:=DO_P_404_START;
   RIO4:1:O.4	:=DO_UV_401_START;
   RIO4:1:O.5	:=DO_RIO4_SPARE_05;
   RIO4:1:O.6	:=DO_RIO4_SPARE_06;
   RIO4:1:O.7	:=DO_RIO4_SPARE_07;
   RIO4:1:O.8	:=DO_RIO4_SPARE_08;
   RIO4:1:O.9	:=DO_RIO4_SPARE_09;
   RIO4:1:O.10	:=DO_RIO4_SPARE_10;
   RIO4:1:O.11	:=DO_RIO4_SPARE_11;
   RIO4:1:O.12	:=DO_RIO4_SPARE_12;
   RIO4:1:O.13	:=DO_RIO4_SPARE_13;
   RIO4:1:O.14	:=DO_RIO4_SPARE_14;
   RIO4:1:O.15	:=DO_RIO4_SPARE_15;
   
   (*ANALOG INPUTS*)
   AI_LIT_401_LEVEL	:=RIO4:2:I.Ch0Data;
   AI_AIT_401_HRDNSS	:=RIO4:2:I.Ch1Data;
   AI_FIT_401_FLOW		:=RIO4:2:I.Ch2Data;
   AI_AIT_402_ORP		:=RIO4:2:I.Ch3Data;
   AI_RIO4_SPARE_03	:=RIO4:2:I.Ch3Data;
   AI_RIO4_SPARE_04	:=RIO4:2:I.Ch4Data;
   AI_RIO4_SPARE_05	:=RIO4:2:I.Ch5Data;
   AI_RIO4_SPARE_06	:=RIO4:2:I.Ch6Data;
   AI_RIO4_SPARE_07	:=RIO4:2:I.Ch7Data;
   AI_RIO4_SPARE_08	:=RIO4:2:I.Ch8Data;
   AI_RIO4_SPARE_09	:=RIO4:2:I.Ch9Data;
   AI_RIO4_SPARE_10	:=RIO4:2:I.Ch10Data;
   AI_RIO4_SPARE_11	:=RIO4:2:I.Ch11Data;
   
   AI_LIT_401_LEVEL_HTY	:=(NOT RIO4:2:I.GeneralFault);
   AI_AIT_401_HRDNSS_HTY	:=(NOT RIO4:2:I.GeneralFault);
   AI_FIT_401_FLOW_HTY		:=(NOT RIO4:2:I.GeneralFault);
   AI_AIT_402_ORP_HTY		:=(NOT RIO4:2:I.GeneralFault);
   AI_RIO4_SPARE_03_HTY	:=(NOT RIO4:2:I.GeneralFault);
   AI_RIO4_SPARE_04_HTY	:=(NOT RIO4:2:I.GeneralFault);
   AI_RIO4_SPARE_05_HTY	:=(NOT RIO4:2:I.GeneralFault);
   AI_RIO4_SPARE_06_HTY	:=(NOT RIO4:2:I.GeneralFault);
   AI_RIO4_SPARE_07_HTY	:=(NOT RIO4:2:I.GeneralFault);
   AI_RIO4_SPARE_08_HTY	:=(NOT RIO4:2:I.GeneralFault);
   AI_RIO4_SPARE_09_HTY	:=(NOT RIO4:2:I.GeneralFault);
   AI_RIO4_SPARE_10_HTY	:=(NOT RIO4:2:I.GeneralFault);
   AI_RIO4_SPARE_11_HTY	:=(NOT RIO4:2:I.GeneralFault);
   
   (*WIRELESS ANALOG INPUTS*)
   W_AI_LIT_401_LEVEL		:=WRIO4:1:I.Ch0Data;
   W_AI_AIT_401_HRDNSS		:=WRIO4:1:I.Ch1Data;
   W_AI_FIT_401_FLOW		:=WRIO4:1:I.Ch2Data;
   W_AI_AIT_402_ORP		:=WRIO4:1:I.Ch3Data;
   
   W_AI_LIT_401_LEVEL_HTY	:=(NOT WRIO4:1:I.Ch0Fault) ;
   W_AI_AIT_401_HRDNSS_HTY	:=(NOT WRIO4:1:I.Ch1Fault) ;
   W_AI_FIT_401_FLOW_HTY	:=(NOT WRIO4:1:I.Ch2Fault) ;
   W_AI_RIO4_SPARE_03_HTY	:=(NOT WRIO4:1:I.Ch3Fault) ;
   
   (*Wireless Selction*)
   HMI_WIFI.PLC_WIFI		:= DI_WIFI_PLC_4;
   HMI_WIFI.RIO_WIFI		:= DI_WIFI_RIO_4;
   
END_ROUTINE

ROUTINE Logix_Status   (* ladder *)
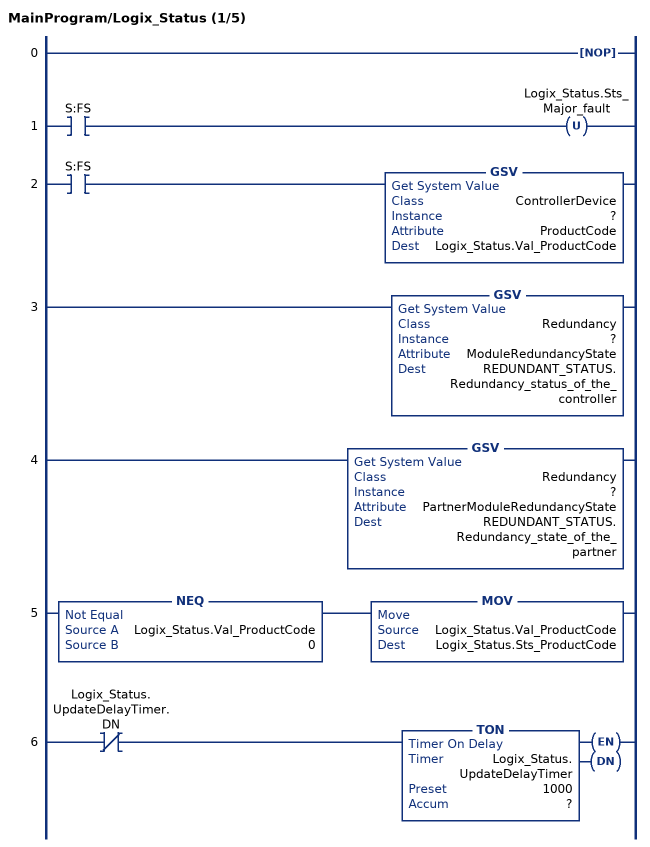
   0: NOP();
   1: XIC(S:FS)OTU(Logix_Status.Sts_Major_fault);
   2: XIC(S:FS)GSV(ControllerDevice,?,ProductCode,Logix_Status.Val_ProductCode);
   3: GSV(Redundancy,?,ModuleRedundancyState,REDUNDANT_STATUS.Redundancy_status_of_the_controller);
   4: GSV(Redundancy,?,PartnerModuleRedundancyState,REDUNDANT_STATUS.Redundancy_state_of_the_partner);
   5: NEQ(Logix_Status.Val_ProductCode,0)MOV(Logix_Status.Val_ProductCode,Logix_Status.Sts_ProductCode);
   6: XIO(Logix_Status.UpdateDelayTimer.DN)TON(Logix_Status.UpdateDelayTimer,?,?);
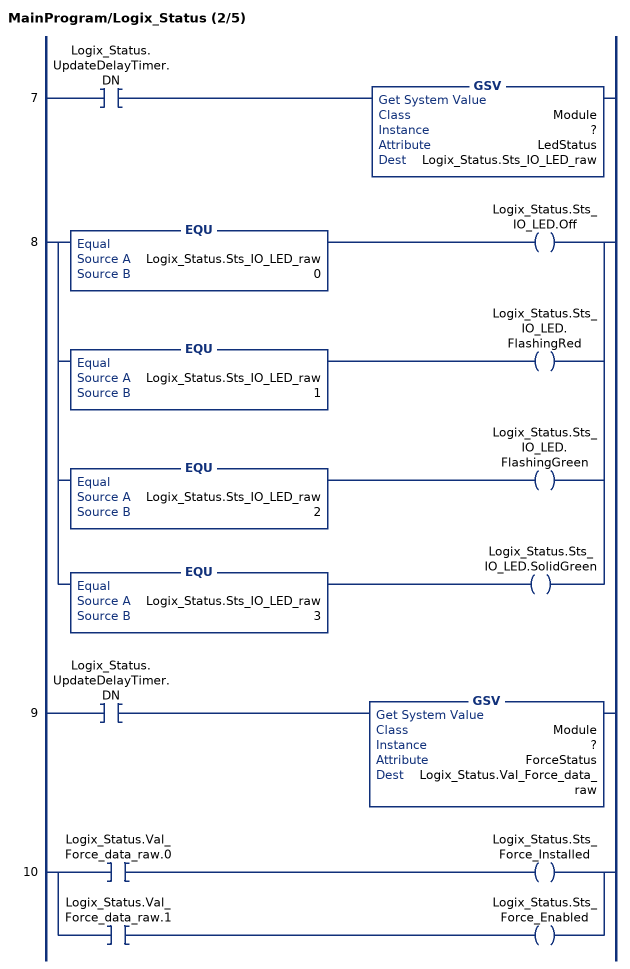
   7: XIC(Logix_Status.UpdateDelayTimer.DN)GSV(Module,?,LedStatus,Logix_Status.Sts_IO_LED_raw);
   8: [EQU(Logix_Status.Sts_IO_LED_raw,0) OTE(Logix_Status.Sts_IO_LED.Off) ,EQU(Logix_Status.Sts_IO_LED_raw,1) OTE(Logix_Status.Sts_IO_LED.FlashingRed) ,EQU(Logix_Status.Sts_IO_LED_raw,2) OTE(Logix_Status.Sts_IO_LED.FlashingGreen) ,EQU(Logix_Status.Sts_IO_LED_raw,3) OTE(Logix_Status.Sts_IO_LED.SolidGreen) ];
   9: XIC(Logix_Status.UpdateDelayTimer.DN)GSV(Module,?,ForceStatus,Logix_Status.Val_Force_data_raw);
   10: [XIC(Logix_Status.Val_Force_data_raw.0) OTE(Logix_Status.Sts_Force_Installed) ,XIC(Logix_Status.Val_Force_data_raw.1) OTE(Logix_Status.Sts_Force_Enabled) ];
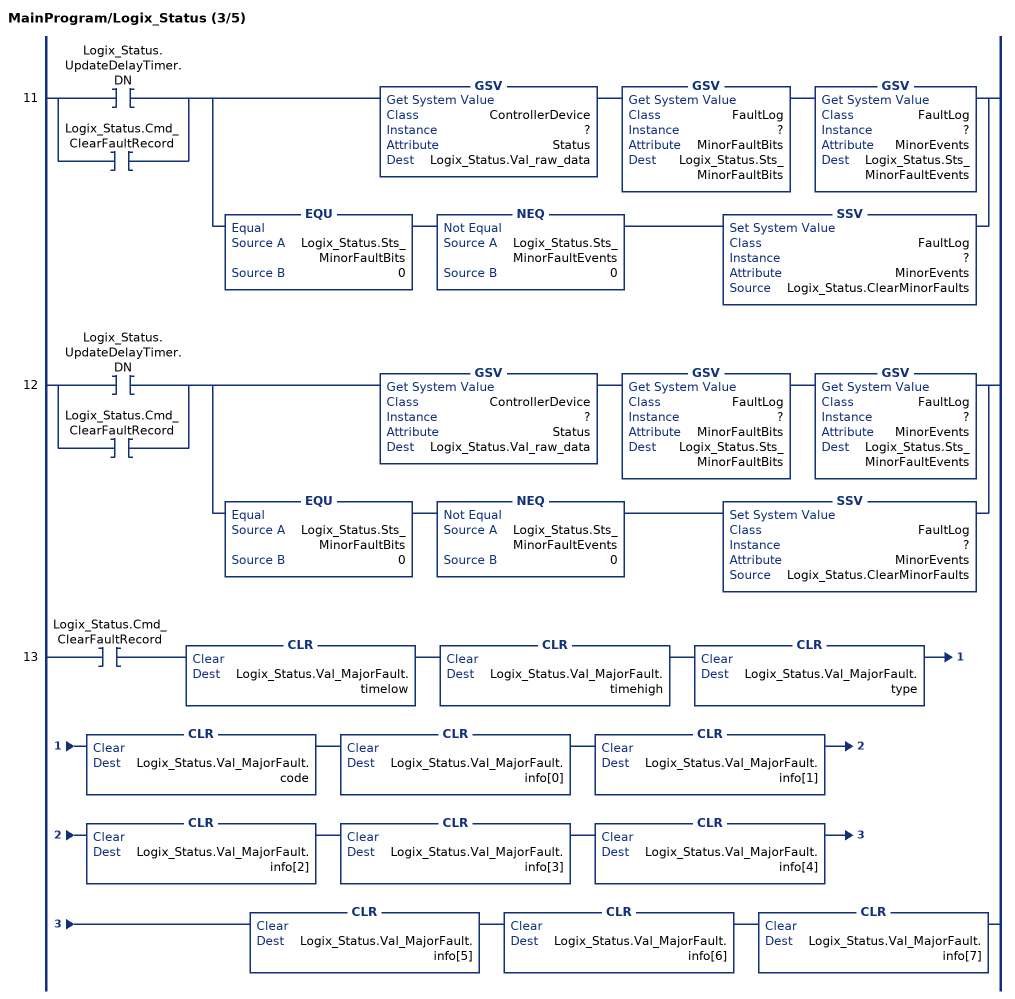
   11: [XIC(Logix_Status.UpdateDelayTimer.DN) ,XIC(Logix_Status.Cmd_ClearFaultRecord) ][GSV(ControllerDevice,?,Status,Logix_Status.Val_raw_data) GSV(FaultLog,?,MinorFaultBits,Logix_Status.Sts_MinorFaultBits) GSV(FaultLog,?,MinorEvents,Logix_Status.Sts_MinorFaultEvents) ,EQU(Logix_Status.Sts_MinorFaultBits,0) NEQ(Logix_Status.Sts_MinorFaultEvents,0) SSV(FaultLog,?,MinorEvents,Logix_Status.ClearMinorFaults) ];
   12: [XIC(Logix_Status.UpdateDelayTimer.DN) ,XIC(Logix_Status.Cmd_ClearFaultRecord) ][GSV(ControllerDevice,?,Status,Logix_Status.Val_raw_data) GSV(FaultLog,?,MinorFaultBits,Logix_Status.Sts_MinorFaultBits) GSV(FaultLog,?,MinorEvents,Logix_Status.Sts_MinorFaultEvents) ,EQU(Logix_Status.Sts_MinorFaultBits,0) NEQ(Logix_Status.Sts_MinorFaultEvents,0) SSV(FaultLog,?,MinorEvents,Logix_Status.ClearMinorFaults) ];
   13: XIC(Logix_Status.Cmd_ClearFaultRecord)CLR(Logix_Status.Val_MajorFault.timelow)CLR(Logix_Status.Val_MajorFault.timehigh)CLR(Logix_Status.Val_MajorFault.type)CLR(Logix_Status.Val_MajorFault.code)CLR(Logix_Status.Val_MajorFault.info[0])CLR(Logix_Status.Val_MajorFault.info[1])CLR(Logix_Status.Val_MajorFault.info[2])CLR(Logix_Status.Val_MajorFault.info[3])CLR(Logix_Status.Val_MajorFault.info[4])CLR(Logix_Status.Val_MajorFault.info[5])CLR(Logix_Status.Val_MajorFault.info[6])CLR(Logix_Status.Val_MajorFault.info[7]);
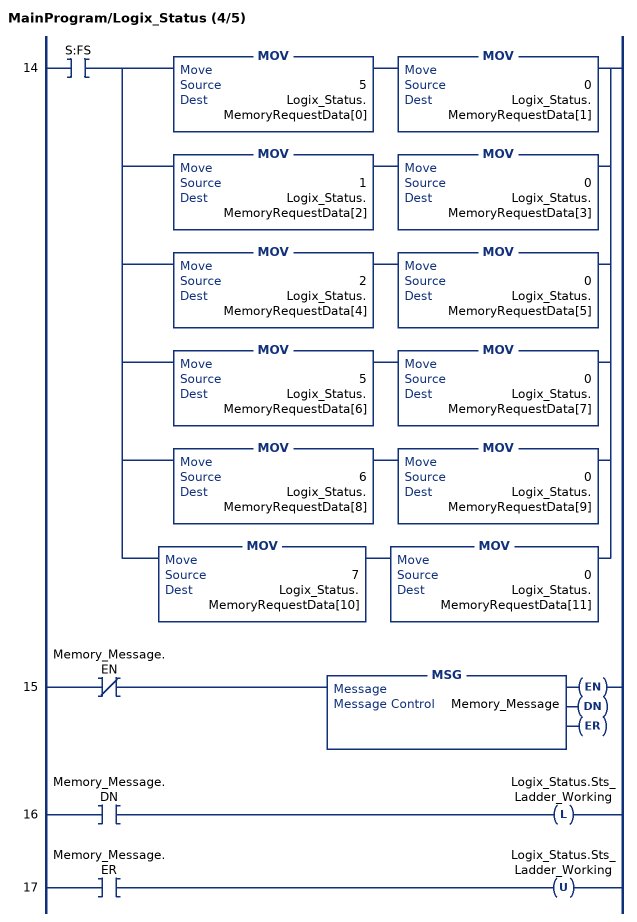
   14: XIC(S:FS)[MOV(5,Logix_Status.MemoryRequestData[0]) MOV(0,Logix_Status.MemoryRequestData[1]) ,MOV(1,Logix_Status.MemoryRequestData[2]) MOV(0,Logix_Status.MemoryRequestData[3]) ,MOV(2,Logix_Status.MemoryRequestData[4]) MOV(0,Logix_Status.MemoryRequestData[5]) ,MOV(5,Logix_Status.MemoryRequestData[6]) MOV(0,Logix_Status.MemoryRequestData[7]) ,MOV(6,Logix_Status.MemoryRequestData[8]) MOV(0,Logix_Status.MemoryRequestData[9]) ,MOV(7,Logix_Status.MemoryRequestData[10]) MOV(0,Logix_Status.MemoryRequestData[11]) ];
   15: XIO(Memory_Message.EN)MSG(Memory_Message);
   16: XIC(Memory_Message.DN)OTL(Logix_Status.Sts_Ladder_Working);
   17: XIC(Memory_Message.ER)OTU(Logix_Status.Sts_Ladder_Working);
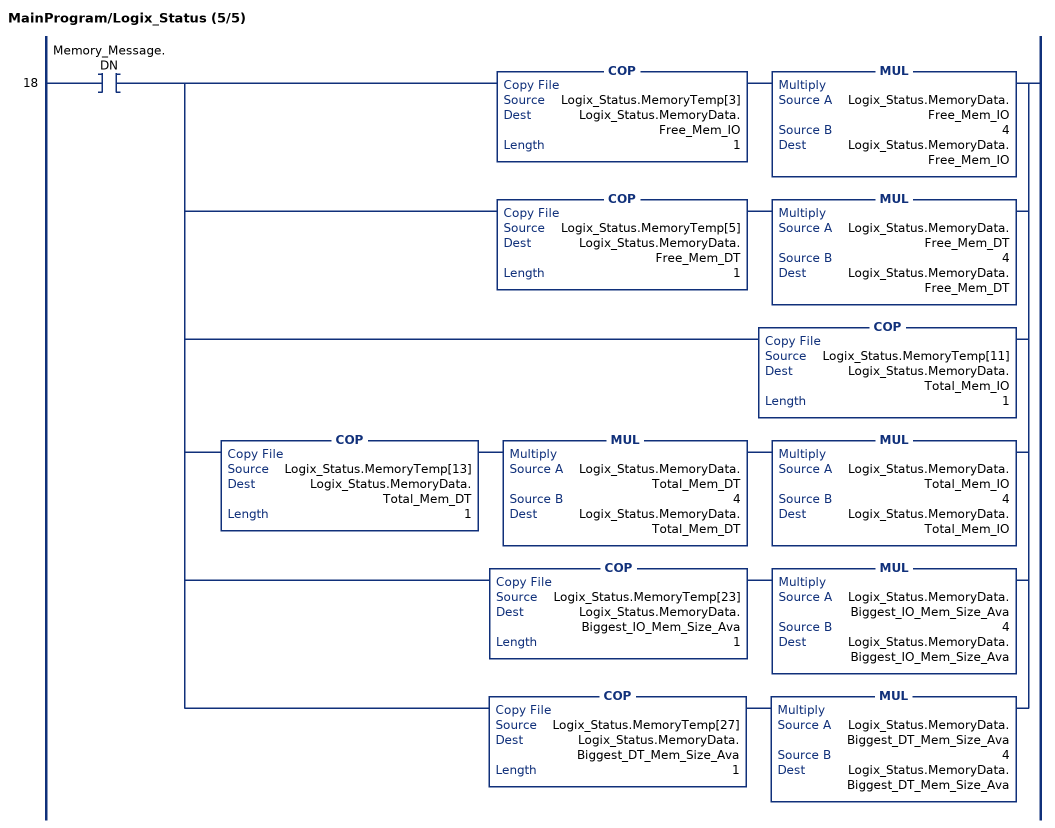
   18: XIC(Memory_Message.DN)[COP(Logix_Status.MemoryTemp[3],Logix_Status.MemoryData.Free_Mem_IO,1) MUL(Logix_Status.MemoryData.Free_Mem_IO,4,Logix_Status.MemoryData.Free_Mem_IO) ,COP(Logix_Status.MemoryTemp[5],Logix_Status.MemoryData.Free_Mem_DT,1) MUL(Logix_Status.MemoryData.Free_Mem_DT,4,Logix_Status.MemoryData.Free_Mem_DT) ,COP(Logix_Status.MemoryTemp[11],Logix_Status.MemoryData.Total_Mem_IO,1) ,COP(Logix_Status.MemoryTemp[13],Logix_Status.MemoryData.Total_Mem_DT,1) MUL(Logix_Status.MemoryData.Total_Mem_DT,4,Logix_Status.MemoryData.Total_Mem_DT) MUL(Logix_Status.MemoryData.Total_Mem_IO,4,Logix_Status.MemoryData.Total_Mem_IO) ,COP(Logix_Status.MemoryTemp[23],Logix_Status.MemoryData.Biggest_IO_Mem_Size_Ava,1) MUL(Logix_Status.MemoryData.Biggest_IO_Mem_Size_Ava,4,Logix_Status.MemoryData.Biggest_IO_Mem_Size_Ava) ,COP(Logix_Status.MemoryTemp[27],Logix_Status.MemoryData.Biggest_DT_Mem_Size_Ava,1) MUL(Logix_Status.MemoryData.Biggest_DT_Mem_Size_Ava,4,Logix_Status.MemoryData.Biggest_DT_Mem_Size_Ava) ];
END_ROUTINE

ROUTINE Main_Seq   (* structured text *)
   (*IF HMI_PLANT.STOP THEN
   	HMI_P4_STATE:=1;
   END_IF;
   *)
   
   (*
   if S:FS then
   	HMI_P4_STATE := 1;
   end_if;
   *)
   
   
   (*-----------WRITE FAULT CONDITION--------------*)
   
   CASE HMI_P4_STATE OF
   	1:(*PLANT IN STANDBY*)
   		_UV401_AutoInp				:=0;
   		_P_RO_FEED_DUTY_AutoInp		:=0;
   		_P_NAHSO3_ORP_DUTY_AutoInp	:=0;
   
   		IF HMI_P4_PERMISSIVE.ON AND HMI_PLANT.START THEN
   			HMI_P4_STATE:=2;
   		END_IF;
   
   	2:(*P401/2 , RO FEED PUMP*)
   		_UV401_AutoInp				:=0;
   		_P_RO_FEED_DUTY_AutoInp		:= HMI_MV503.STATUS=2 AND HMI_MV504.STATUS=2 ;
   		_P_NAHSO3_ORP_DUTY_AutoInp	:=0;
   
   		IF HMI_P_RO_FEED_DUTY.Pump_Running THEN
   			HMI_P4_STATE:=3;
   		END_IF;
   
   
   	3:(*UV401, DECHLORINATION UV*)
   		_UV401_AutoInp				:=1;
   		_P_RO_FEED_DUTY_AutoInp		:=1;
   		_P_NAHSO3_ORP_DUTY_AutoInp	:=0;
   
   		IF HMI_UV401.Status=2 THEN
   			HMI_P4_STATE:=4;
   		END_IF;
   
   	4:(*P403/4 , NAHSO4*)
   		_UV401_AutoInp				:=1;
   		_P_RO_FEED_DUTY_AutoInp		:=1;
   
   		_P_NAHSO3_ORP_DUTY_SR.EnableIn		:= 1;
   		_P_NAHSO3_ORP_DUTY_SR.Set			:= (HMI_P401.Status=2 OR HMI_P402.Status=2) AND (HMI_AIT402.AH);
   		_P_NAHSO3_ORP_DUTY_SR.Reset			:= (HMI_P401.Status<>2 AND HMI_P402.Status<>2) OR (HMI_AIT402.AL);
   		SETD(_P_NAHSO3_ORP_DUTY_SR);
   		_P_NAHSO3_ORP_DUTY_AutoInp			:= _P_NAHSO3_ORP_DUTY_SR.Out;
   
   		IF HMI_RO_HPP_SD.ON THEN
   			HMI_P4_STATE:=5;
   		END_IF;
   
   	5:(*SHUTDOWN RO FEED*)
   		_UV401_AutoInp				:=1;
   		_P_RO_FEED_DUTY_AutoInp		:=HMI_MV503.STATUS=1 AND HMI_MV504.STATUS=1;
   		_P_NAHSO3_ORP_DUTY_AutoInp	:= 0;;
   
   		IF NOT HMI_P_RO_FEED_DUTY.Pump_Running THEN
   			HMI_P4_STATE:=6;
   		END_IF;
   
   	6:(*SHUTDOWN UV*)
   		_UV401_AutoInp				:=0;
   		_P_RO_FEED_DUTY_AutoInp		:=0;
   		_P_NAHSO3_ORP_DUTY_AutoInp	:= 0;
   
   		IF HMI_UV401.STATUS=1 THEN
   			HMI_P4_STATE:=1;
   		END_IF;
   ELSE
   	HMI_P4_STATE:=1;
   END_CASE;
   
   
   
   
   
   
   
   
   
   
   
   
   
   
   
   
   
   
   
   
END_ROUTINE

ROUTINE MainRoutine   (* ladder *)
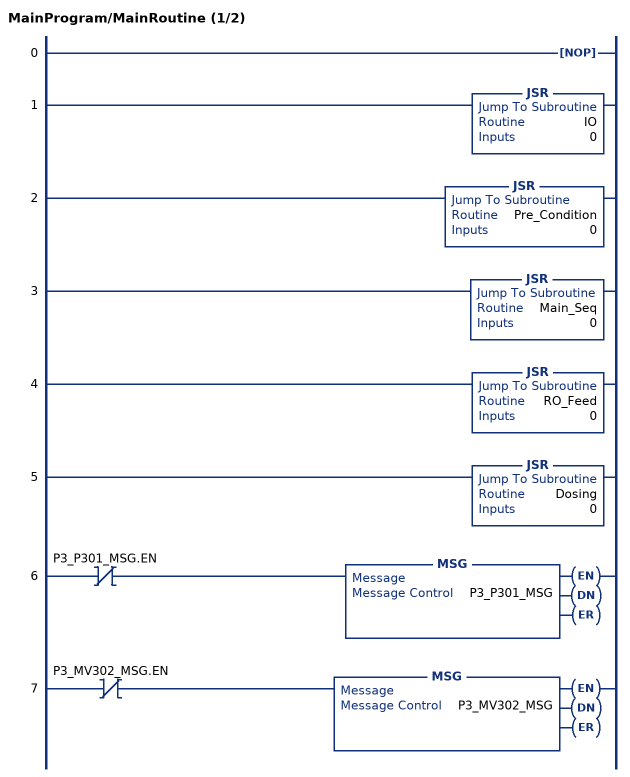
   0: NOP();
   1: JSR(IO,0);
   2: JSR(Pre_Condition,0);
   3: JSR(Main_Seq,0);
   4: JSR(RO_Feed,0);
   5: JSR(Dosing,0);
   6: XIO(P3_P301_MSG.EN)MSG(P3_P301_MSG);
   7: XIO(P3_MV302_MSG.EN)MSG(P3_MV302_MSG);
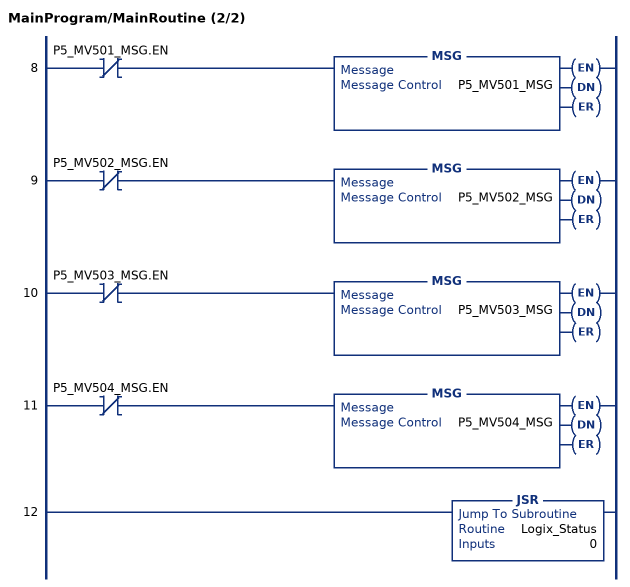
   8: XIO(P5_MV501_MSG.EN)MSG(P5_MV501_MSG);
   9: XIO(P5_MV502_MSG.EN)MSG(P5_MV502_MSG);
   10: XIO(P5_MV503_MSG.EN)MSG(P5_MV503_MSG);
   11: XIO(P5_MV504_MSG.EN)MSG(P5_MV504_MSG);
   12: JSR(Logix_Status,0);
END_ROUTINE

ROUTINE Pre_Condition   (* structured text *)
   (*RESET ALL INSTRUMENT*)
   IF HMI_PLANT_RESET.ON THEN
   	HMI_P401.Reset	:=1;
   	HMI_P402.Reset	:=1;
   	HMI_P403.Reset	:=1;
   	HMI_P404.Reset	:=1;
   	HMI_UV401.Reset	:=1;
   END_IF;
   
   (*ALL INSTRUMENT IN AUTO MODE*)
   IF HMI_PLANT_AUTO.ON THEN
   	HMI_P401.Auto	:=1;
   	HMI_P402.Auto	:=1;
   	HMI_P403.Auto	:=1;
   	HMI_P404.Auto	:=1;
   	HMI_UV401.Auto	:=1;
   END_IF;
   
   (*ALL INSTRUMENT IN MANUAL MODE*)
   IF HMI_PLANT_AUTO.OFF THEN
   	HMI_P401.Auto	:=0;
   	HMI_P402.Auto	:=0;
   	HMI_P403.Auto	:=0;
   	HMI_P404.Auto	:=0;
   	HMI_UV401.Auto	:=0;
   END_IF;
   
   HMI_P4_PERMISSIVE.ON:= (HMI_P401.Avl OR HMI_P402.Avl) AND (HMI_P403.Avl OR HMI_P404.Avl) AND HMI_UV401.AVL;
   
   (*Enable Flow Totalising*)
   _FIT401_Tot_Enb	:= HMI_P401.status=2 OR HMI_P402.status=2;
   
   TON_FIT401_TM.PRE 			:= 	6*1000;
   TON_FIT401_TM.TimerEnable 	:=  (HMI_P401.STATUS=2 OR HMI_P402.STATUS=2 )AND HMI_FIT401.ALL;
   TONR(TON_FIT401_TM);
   
   TON_FIT401_P1_TM.PRE 			:= 	6*1000;
   TON_FIT401_P1_TM.TimerEnable 	:=  HMI_FIT401.ALL AND HMI_P401.STATUS=2;
   TONR(TON_FIT401_P1_TM);
   
   TON_FIT401_P2_TM.PRE 			:= 	6*1000;
   TON_FIT401_P2_TM.TimerEnable 	:=  HMI_FIT401.ALL AND HMI_P402.STATUS=2;
   TONR(TON_FIT401_P2_TM);
   
   (*P401 Permissive*)
   HMI_P401.Permissive.0 	:= NOT HMI_LIT401.ALL;
   HMI_P401.Permissive.1 	:= HMI_MV501.STATUS=2 OR HMI_MV502.STATUS=2 OR HMI_MV503.STATUS=2 OR HMI_MV504.STATUS=2 ;
   HMI_P401.Permissive.2 	:= 1;
   HMI_P401.Permissive.3 	:= 1;
   HMI_P401.Permissive.4 	:= 1;
   HMI_P401.Permissive.5 	:= 1;
   HMI_P401.Permissive.6 	:= 1;
   HMI_P401.Permissive.7 	:= 1;
   HMI_P401.Permissive.8 	:= 1;
   HMI_P401.Permissive.9 	:= 1;
   HMI_P401.Permissive.10 	:= 1;
   HMI_P401.Permissive.11 	:= 1;
   HMI_P401.Permissive.12 	:= 1;
   HMI_P401.Permissive.13	:= 1;
   HMI_P401.Permissive.14	:= 1;
   HMI_P401.Permissive.15 	:= 1;
   
   HMI_P401_MSG.PERMISSIVE1 := HMI_P401.Permissive.0;
   HMI_P401_MSG.PERMISSIVE2 := 0;
   HMI_P401_MSG.PERMISSIVE3 := 0;
   HMI_P401_MSG.PERMISSIVE4 := 0;
   HMI_P401_MSG.PERMISSIVE5 := 0;
   
   (*P402 Permissive*)
   HMI_P402.Permissive.0 	:= NOT HMI_LIT401.ALL;
   HMI_P402.Permissive.1 	:= HMI_MV501.STATUS=2 OR HMI_MV502.STATUS=2 OR HMI_MV503.STATUS=2 OR HMI_MV504.STATUS=2 ;
   HMI_P402.Permissive.2 	:= 1;
   HMI_P402.Permissive.3 	:= 1;
   HMI_P402.Permissive.4 	:= 1;
   HMI_P402.Permissive.5 	:= 1;
   HMI_P402.Permissive.6 	:= 1;
   HMI_P402.Permissive.7 	:= 1;
   HMI_P402.Permissive.8 	:= 1;
   HMI_P402.Permissive.9 	:= 1;
   HMI_P402.Permissive.10 	:= 1;
   HMI_P402.Permissive.11 	:= 1;
   HMI_P402.Permissive.12 	:= 1;
   HMI_P402.Permissive.13	:= 1;
   HMI_P402.Permissive.14	:= 1;
   HMI_P402.Permissive.15 	:= 1;
   
   HMI_P402_MSG.PERMISSIVE1 := HMI_P402.Permissive.0;
   HMI_P402_MSG.PERMISSIVE2 := 0;
   HMI_P402_MSG.PERMISSIVE3 := 0;
   HMI_P402_MSG.PERMISSIVE4 := 0;
   HMI_P402_MSG.PERMISSIVE5 := 0;
   
   (*P403 Permissive*)
   HMI_P403.Permissive.0 	:= NOT HMI_LS401.ALARM;
   HMI_P403.Permissive.1 	:= HMI_P401.STATUS=2 OR HMI_P402.STATUS=2;
   HMI_P403.Permissive.2 	:= 1;
   HMI_P403.Permissive.3 	:= 1;
   HMI_P403.Permissive.4 	:= 1;
   HMI_P403.Permissive.5 	:= 1;
   HMI_P403.Permissive.6 	:= 1;
   HMI_P403.Permissive.7 	:= 1;
   HMI_P403.Permissive.8 	:= 1;
   HMI_P403.Permissive.9 	:= 1;
   HMI_P403.Permissive.10 	:= 1;
   HMI_P403.Permissive.11 	:= 1;
   HMI_P403.Permissive.12 	:= 1;
   HMI_P403.Permissive.13	:= 1;
   HMI_P403.Permissive.14	:= 1;
   HMI_P403.Permissive.15 	:= 1;
   
   HMI_P403_MSG.PERMISSIVE1 := HMI_P403.Permissive.0;
   HMI_P403_MSG.PERMISSIVE2 := HMI_P403.Permissive.1;
   HMI_P403_MSG.PERMISSIVE3 := 0;
   HMI_P403_MSG.PERMISSIVE4 := 0;
   HMI_P403_MSG.PERMISSIVE5 := 0;
   
   
   (*P404 Permissive*)
   HMI_P404.Permissive.0 	:= NOT HMI_LS401.ALARM;
   HMI_P404.Permissive.1 	:= HMI_P401.STATUS=2 OR HMI_P402.STATUS=2;
   HMI_P404.Permissive.2 	:= 1;
   HMI_P404.Permissive.3 	:= 1;
   HMI_P404.Permissive.4 	:= 1;
   HMI_P404.Permissive.5 	:= 1;
   HMI_P404.Permissive.6 	:= 1;
   HMI_P404.Permissive.7 	:= 1;
   HMI_P404.Permissive.8 	:= 1;
   HMI_P404.Permissive.9 	:= 1;
   HMI_P404.Permissive.10 	:= 1;
   HMI_P404.Permissive.11 	:= 1;
   HMI_P404.Permissive.12 	:= 1;
   HMI_P404.Permissive.13	:= 1;
   HMI_P404.Permissive.14	:= 1;
   HMI_P404.Permissive.15 	:= 1;
   
   HMI_P404_MSG.PERMISSIVE1 := HMI_P404.Permissive.0;
   HMI_P404_MSG.PERMISSIVE2 := HMI_P404.Permissive.1;
   HMI_P404_MSG.PERMISSIVE3 := 0;
   HMI_P404_MSG.PERMISSIVE4 := 0;
   HMI_P404_MSG.PERMISSIVE5 := 0;
   
   (*UV401 Permissive*)
   HMI_UV401.Permissive.0 	:= HMI_P401.STATUS=2 OR HMI_P402.STATUS=2;
   HMI_UV401.Permissive.1 	:= NOT HMI_FIT401.ALL;
   HMI_UV401.Permissive.2 	:= 1;
   HMI_UV401.Permissive.3 	:= 1;
   HMI_UV401.Permissive.4 	:= 1;
   HMI_UV401.Permissive.5 	:= 1;
   HMI_UV401.Permissive.6 	:= 1;
   HMI_UV401.Permissive.7 	:= 1;
   HMI_UV401.Permissive.8 	:= 1;
   HMI_UV401.Permissive.9 	:= 1;
   HMI_UV401.Permissive.10 := 1;
   HMI_UV401.Permissive.11 := 1;
   HMI_UV401.Permissive.12 := 1;
   HMI_UV401.Permissive.13	:= 1;
   HMI_UV401.Permissive.14	:= 1;
   HMI_UV401.Permissive.15 := 1;
   
   HMI_UV401_MSG.PERMISSIVE1 := HMI_P403.Permissive.0;
   HMI_UV401_MSG.PERMISSIVE2 := HMI_P403.Permissive.1;
   HMI_UV401_MSG.PERMISSIVE3 := 0;
   HMI_UV401_MSG.PERMISSIVE4 := 0;
   HMI_UV401_MSG.PERMISSIVE5 := 0;
   
   (*-------------------------------------------------------------------------------------*)
   (*P401 Shutdown*)
   HMI_P401.SD.0 	:= HMI_LIT401.ALL;
   HMI_P401.SD.1 	:= TON_FIT401_P1_TM.DN;
   HMI_P401.SD.2 	:= HMI_P401.STATUS=2 AND HMI_MV501.STATUS<>2 AND HMI_MV502.STATUS<>2 AND HMI_MV503.STATUS<>2 AND HMI_MV504.STATUS<>2 ;
   HMI_P401.SD.3 	:= 0;
   HMI_P401.SD.4 	:= 0;
   HMI_P401.SD.5 	:= 0;
   HMI_P401.SD.6 	:= 0;
   HMI_P401.SD.7 	:= 0;
   HMI_P401.SD.8 	:= 0;
   HMI_P401.SD.9 	:= 0;
   HMI_P401.SD.10 	:= 0;
   HMI_P401.SD.11 	:= 0;
   HMI_P401.SD.12 	:= 0;
   HMI_P401.SD.13 	:= 0;
   HMI_P401.SD.14 	:= 0;
   HMI_P401.SD.15 	:= 0;
   
   HMI_P401_MSG.SHUTDOWN1 := HMI_P401.SHUTDOWN.0 ;
   HMI_P401_MSG.SHUTDOWN2 := HMI_P401.SHUTDOWN.1 ;
   HMI_P401_MSG.SHUTDOWN3 := HMI_P401.SHUTDOWN.2 ;
   HMI_P401_MSG.SHUTDOWN4 := HMI_P401.SHUTDOWN.3 ;
   HMI_P401_MSG.SHUTDOWN5 := HMI_P401.SHUTDOWN.4 ;
   
   (*P402 Shutdown*)
   HMI_P402.SD.0 	:= HMI_LIT401.ALL;
   HMI_P402.SD.1 	:= TON_FIT401_P2_TM.DN;
   HMI_P402.SD.2 	:= HMI_P402.STATUS=2 AND HMI_MV501.STATUS<>2 AND HMI_MV502.STATUS<>2 AND HMI_MV503.STATUS<>2 AND HMI_MV504.STATUS<>2 ;
   HMI_P402.SD.3 	:= 0;
   HMI_P402.SD.4 	:= 0;
   HMI_P402.SD.5 	:= 0;
   HMI_P402.SD.6 	:= 0;
   HMI_P402.SD.7 	:= 0;
   HMI_P402.SD.8 	:= 0;
   HMI_P402.SD.9 	:= 0;
   HMI_P402.SD.10 	:= 0;
   HMI_P402.SD.11 	:= 0;
   HMI_P402.SD.12 	:= 0;
   HMI_P402.SD.13 	:= 0;
   HMI_P402.SD.14 	:= 0;
   HMI_P402.SD.15 	:= 0;
   
   HMI_P402_MSG.SHUTDOWN1 := HMI_P402.SHUTDOWN.0 ;
   HMI_P402_MSG.SHUTDOWN2 := HMI_P402.SHUTDOWN.1 ;
   HMI_P402_MSG.SHUTDOWN3 := HMI_P402.SHUTDOWN.2 ;
   HMI_P402_MSG.SHUTDOWN4 := HMI_P402.SHUTDOWN.3 ;
   HMI_P402_MSG.SHUTDOWN5 := HMI_P402.SHUTDOWN.4 ;
   
   (*P403 Shutdown*)
   HMI_P403.SD.0 	:= HMI_LS401.ALARM;
   HMI_P403.SD.1 	:= (HMI_P401.STATUS=2 OR HMI_P402.STATUS=2 )AND HMI_FIT401.ALL;
   HMI_P403.SD.2 	:= 0;
   HMI_P403.SD.3 	:= 0;
   HMI_P403.SD.4 	:= 0;
   HMI_P403.SD.5 	:= 0;
   HMI_P403.SD.6 	:= 0;
   HMI_P403.SD.7 	:= 0;
   HMI_P403.SD.8 	:= 0;
   HMI_P403.SD.9 	:= 0;
   HMI_P403.SD.10 	:= 0;
   HMI_P403.SD.11 	:= 0;
   HMI_P403.SD.12 	:= 0;
   HMI_P403.SD.13 	:= 0;
   HMI_P403.SD.14 	:= 0;
   HMI_P403.SD.15 	:= 0;
   
   HMI_P403_MSG.SHUTDOWN1 := HMI_P403.SHUTDOWN.0 ;
   HMI_P403_MSG.SHUTDOWN2 := HMI_P403.SHUTDOWN.1 ;
   HMI_P403_MSG.SHUTDOWN3 := HMI_P403.SHUTDOWN.2 ;
   HMI_P403_MSG.SHUTDOWN4 := HMI_P403.SHUTDOWN.3 ;
   HMI_P403_MSG.SHUTDOWN5 := HMI_P403.SHUTDOWN.4 ;
   
   (*P404 Shutdown*)
   HMI_P404.SD.0 	:= HMI_LS401.ALARM;
   HMI_P404.SD.1 	:= (HMI_P401.STATUS=2 OR HMI_P402.STATUS=2) AND HMI_FIT401.ALL;
   HMI_P404.SD.2 	:= 0;
   HMI_P404.SD.3 	:= 0;
   HMI_P404.SD.4 	:= 0;
   HMI_P404.SD.5 	:= 0;
   HMI_P404.SD.6 	:= 0;
   HMI_P404.SD.7 	:= 0;
   HMI_P404.SD.8 	:= 0;
   HMI_P404.SD.9 	:= 0;
   HMI_P404.SD.10 	:= 0;
   HMI_P404.SD.11 	:= 0;
   HMI_P404.SD.12 	:= 0;
   HMI_P404.SD.13 	:= 0;
   HMI_P404.SD.14 	:= 0;
   HMI_P404.SD.15 	:= 0;
   
   HMI_P404_MSG.SHUTDOWN1 := HMI_P404.SHUTDOWN.0 ;
   HMI_P404_MSG.SHUTDOWN2 := HMI_P404.SHUTDOWN.1 ;
   HMI_P404_MSG.SHUTDOWN3 := HMI_P404.SHUTDOWN.2 ;
   HMI_P404_MSG.SHUTDOWN4 := HMI_P404.SHUTDOWN.3 ;
   HMI_P404_MSG.SHUTDOWN5 := HMI_P404.SHUTDOWN.4 ;
   
   (*UV401 Shutdown*)
   HMI_UV401.SD.0 	:= TON_FIT401_TM.DN;
   HMI_UV401.SD.1 	:= 0;
   HMI_UV401.SD.2 	:= 0;
   HMI_UV401.SD.3 	:= 0;
   HMI_UV401.SD.4 	:= 0;
   HMI_UV401.SD.5 	:= 0;
   HMI_UV401.SD.6 	:= 0;
   HMI_UV401.SD.7 	:= 0;
   HMI_UV401.SD.8 	:= 0;
   HMI_UV401.SD.9 	:= 0;
   HMI_UV401.SD.10 	:= 0;
   HMI_UV401.SD.11 	:= 0;
   HMI_UV401.SD.12 	:= 0;
   HMI_UV401.SD.13 	:= 0;
   HMI_UV401.SD.14 	:= 0;
   HMI_UV401.SD.15 	:= 0;
   
   HMI_UV401_MSG.SHUTDOWN1 := HMI_UV401.SHUTDOWN.0 ;
   HMI_UV401_MSG.SHUTDOWN2 := HMI_UV401.SHUTDOWN.1 ;
   HMI_UV401_MSG.SHUTDOWN3 := HMI_UV401.SHUTDOWN.2 ;
   HMI_UV401_MSG.SHUTDOWN4 := HMI_UV401.SHUTDOWN.3 ;
   HMI_UV401_MSG.SHUTDOWN5 := HMI_UV401.SHUTDOWN.4 ;
   
   
   
   
END_ROUTINE

ROUTINE RO_Feed   (* function block diagram *)
   SHEET 1
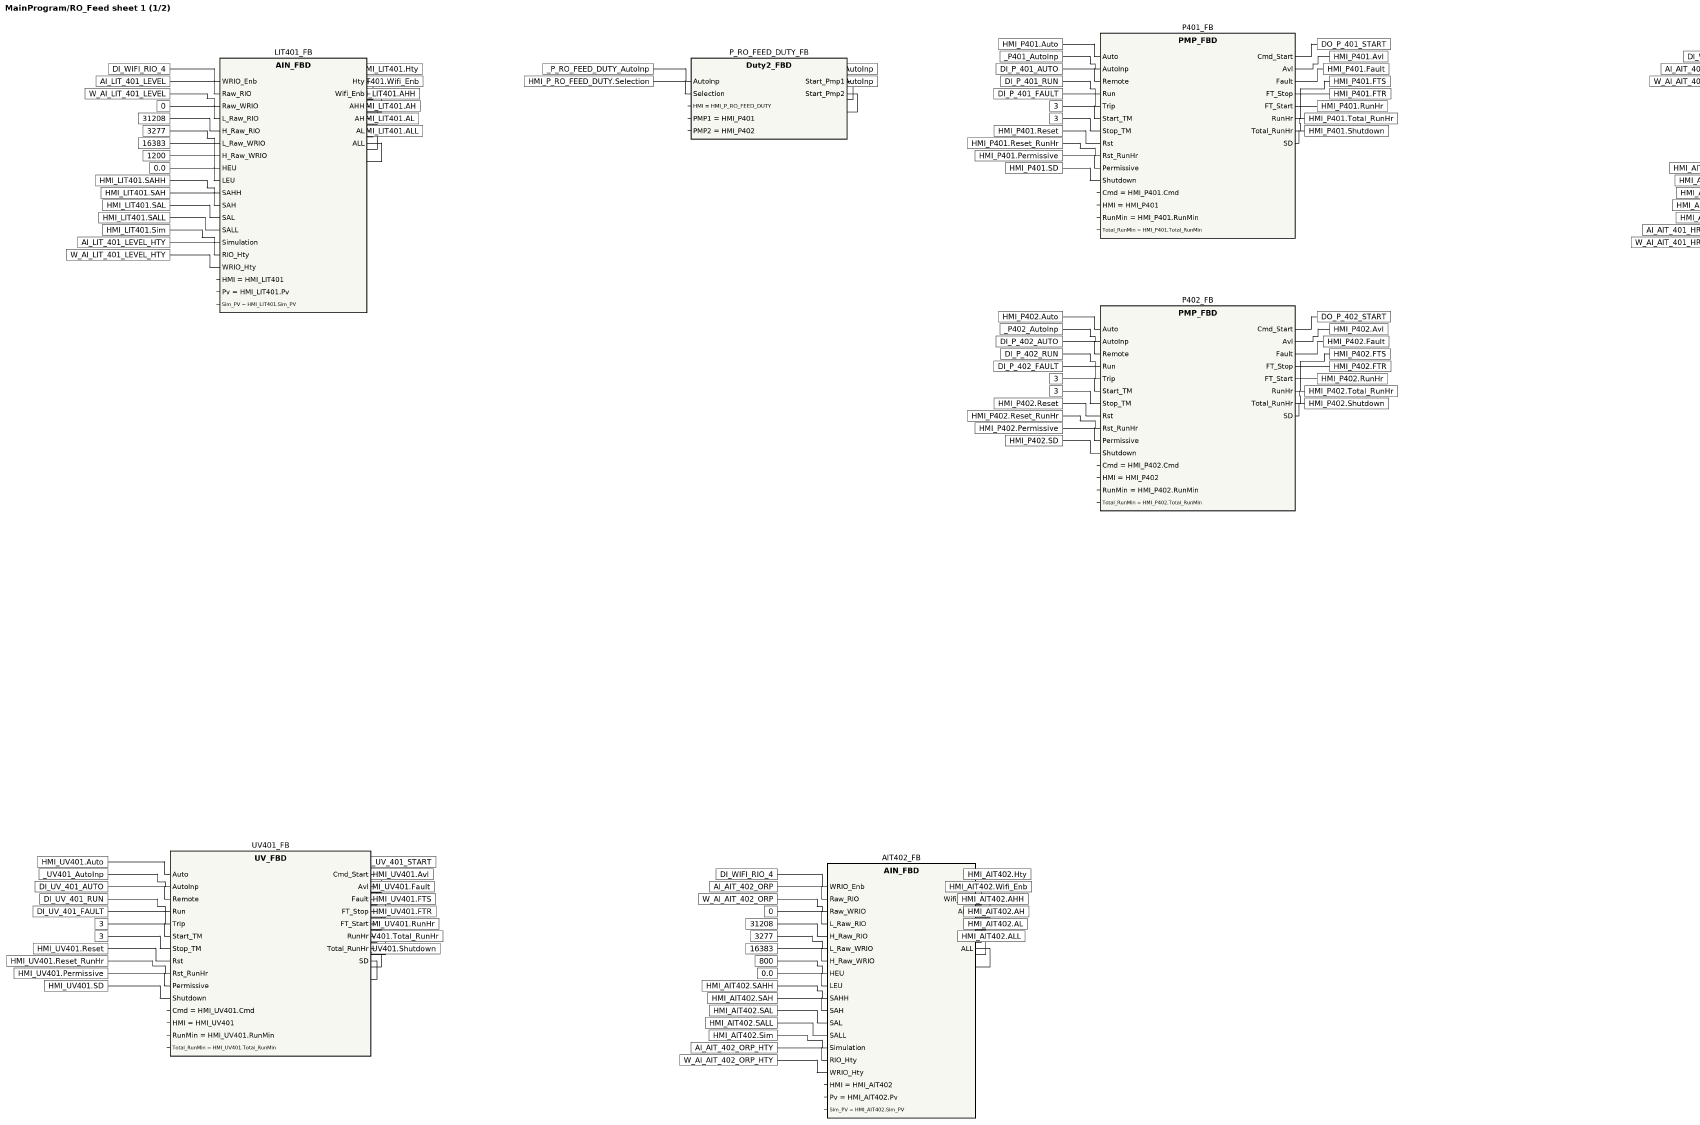
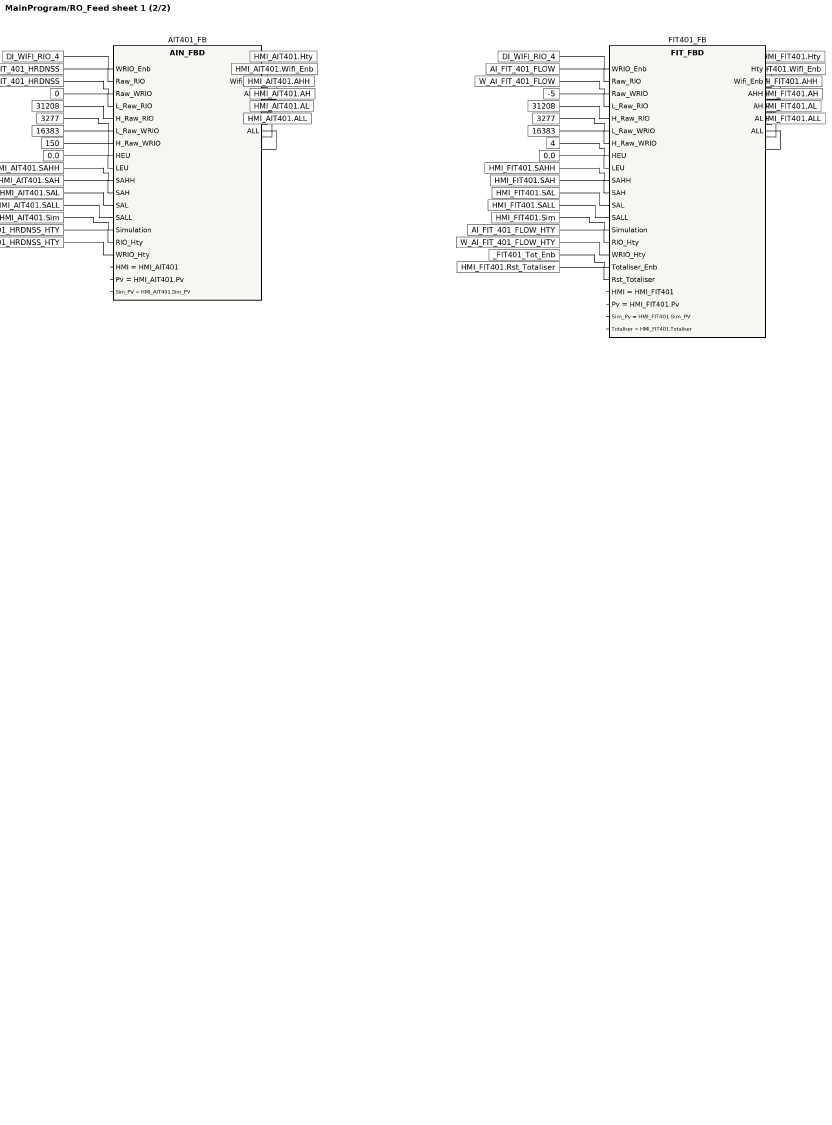
   UV401_FB : UV_FBD(Auto := HMI_UV401.Auto, AutoInp := _UV401_AutoInp, Remote := DI_UV_401_AUTO, Run := DI_UV_401_RUN, Trip := DI_UV_401_FAULT, Start_TM := 3, Stop_TM := 3, Rst := HMI_UV401.Reset, Rst_RunHr := HMI_UV401.Reset_RunHr, Permissive := HMI_UV401.Permissive, Shutdown := HMI_UV401.SD, Cmd := HMI_UV401.Cmd, HMI := HMI_UV401, RunMin := HMI_UV401.RunMin, Total_RunMin := HMI_UV401.Total_RunMin);
   LIT401_FB : AIN_FBD(WRIO_Enb := DI_WIFI_RIO_4, Raw_RIO := AI_LIT_401_LEVEL, Raw_WRIO := W_AI_LIT_401_LEVEL, L_Raw_RIO := 0, H_Raw_RIO := 31208, L_Raw_WRIO := 3277, H_Raw_WRIO := 16383, HEU := 1200, LEU := 0.0, SAHH := HMI_LIT401.SAHH, SAH := HMI_LIT401.SAH, SAL := HMI_LIT401.SAL, SALL := HMI_LIT401.SALL, Simulation := HMI_LIT401.Sim, RIO_Hty := AI_LIT_401_LEVEL_HTY, WRIO_Hty := W_AI_LIT_401_LEVEL_HTY, HMI := HMI_LIT401, Pv := HMI_LIT401.Pv, Sim_PV := HMI_LIT401.Sim_PV);
   HMI_LIT401.Wifi_Enb := LIT401_FB.Wifi_Enb;
   HMI_UV401.Total_RunHr := UV401_FB.Total_RunHr;
   HMI_LIT401.AHH := LIT401_FB.AHH;
   HMI_UV401.Shutdown := UV401_FB.SD;
   HMI_LIT401.Hty := LIT401_FB.Hty;
   HMI_LIT401.AH := LIT401_FB.AH;
   HMI_LIT401.AL := LIT401_FB.AL;
   HMI_LIT401.ALL := LIT401_FB.ALL;
   DO_UV_401_START := UV401_FB.Cmd_Start;
   HMI_UV401.Fault := UV401_FB.Fault;
   HMI_UV401.RunHr := UV401_FB.RunHr;
   HMI_UV401.Avl := UV401_FB.Avl;
   HMI_UV401.FTS := UV401_FB.FT_Stop;
   HMI_UV401.FTR := UV401_FB.FT_Start;
   P_RO_FEED_DUTY_FB : Duty2_FBD(AutoInp := _P_RO_FEED_DUTY_AutoInp, Selection := HMI_P_RO_FEED_DUTY.Selection, HMI := HMI_P_RO_FEED_DUTY, PMP1 := HMI_P401, PMP2 := HMI_P402);
   _P401_AutoInp := P_RO_FEED_DUTY_FB.Start_Pmp1;
   _P402_AutoInp := P_RO_FEED_DUTY_FB.Start_Pmp2;
   AIT402_FB : AIN_FBD(WRIO_Enb := DI_WIFI_RIO_4, Raw_RIO := AI_AIT_402_ORP, Raw_WRIO := W_AI_AIT_402_ORP, L_Raw_RIO := 0, H_Raw_RIO := 31208, L_Raw_WRIO := 3277, H_Raw_WRIO := 16383, HEU := 800, LEU := 0.0, SAHH := HMI_AIT402.SAHH, SAH := HMI_AIT402.SAH, SAL := HMI_AIT402.SAL, SALL := HMI_AIT402.SALL, Simulation := HMI_AIT402.Sim, RIO_Hty := AI_AIT_402_ORP_HTY, WRIO_Hty := W_AI_AIT_402_ORP_HTY, HMI := HMI_AIT402, Pv := HMI_AIT402.Pv, Sim_PV := HMI_AIT402.Sim_PV);
   HMI_AIT402.Wifi_Enb := AIT402_FB.Wifi_Enb;
   HMI_AIT402.AHH := AIT402_FB.AHH;
   HMI_AIT402.ALL := AIT402_FB.ALL;
   HMI_AIT402.Hty := AIT402_FB.Hty;
   HMI_AIT402.AH := AIT402_FB.AH;
   HMI_AIT402.AL := AIT402_FB.AL;
   P401_FB : PMP_FBD(Auto := HMI_P401.Auto, AutoInp := _P401_AutoInp, Remote := DI_P_401_AUTO, Run := DI_P_401_RUN, Trip := DI_P_401_FAULT, Start_TM := 3, Stop_TM := 3, Rst := HMI_P401.Reset, Rst_RunHr := HMI_P401.Reset_RunHr, Permissive := HMI_P401.Permissive, Shutdown := HMI_P401.SD, Cmd := HMI_P401.Cmd, HMI := HMI_P401, RunMin := HMI_P401.RunMin, Total_RunMin := HMI_P401.Total_RunMin);
   P402_FB : PMP_FBD(Auto := HMI_P402.Auto, AutoInp := _P402_AutoInp, Remote := DI_P_402_AUTO, Run := DI_P_402_RUN, Trip := DI_P_402_FAULT, Start_TM := 3, Stop_TM := 3, Rst := HMI_P402.Reset, Rst_RunHr := HMI_P402.Reset_RunHr, Permissive := HMI_P402.Permissive, Shutdown := HMI_P402.SD, Cmd := HMI_P402.Cmd, HMI := HMI_P402, RunMin := HMI_P402.RunMin, Total_RunMin := HMI_P402.Total_RunMin);
   HMI_P401.Total_RunHr := P401_FB.Total_RunHr;
   HMI_P401.Shutdown := P401_FB.SD;
   HMI_P402.Total_RunHr := P402_FB.Total_RunHr;
   HMI_P402.Shutdown := P402_FB.SD;
   DO_P_401_START := P401_FB.Cmd_Start;
   HMI_P401.RunHr := P401_FB.RunHr;
   DO_P_402_START := P402_FB.Cmd_Start;
   HMI_P402.RunHr := P402_FB.RunHr;
   HMI_P401.Fault := P401_FB.Fault;
   HMI_P402.Fault := P402_FB.Fault;
   HMI_P401.Avl := P401_FB.Avl;
   HMI_P401.FTS := P401_FB.FT_Stop;
   HMI_P401.FTR := P401_FB.FT_Start;
   HMI_P402.Avl := P402_FB.Avl;
   HMI_P402.FTS := P402_FB.FT_Stop;
   HMI_P402.FTR := P402_FB.FT_Start;
   AIT401_FB : AIN_FBD(WRIO_Enb := DI_WIFI_RIO_4, Raw_RIO := AI_AIT_401_HRDNSS, Raw_WRIO := W_AI_AIT_401_HRDNSS, L_Raw_RIO := 0, H_Raw_RIO := 31208, L_Raw_WRIO := 3277, H_Raw_WRIO := 16383, HEU := 150, LEU := 0.0, SAHH := HMI_AIT401.SAHH, SAH := HMI_AIT401.SAH, SAL := HMI_AIT401.SAL, SALL := HMI_AIT401.SALL, Simulation := HMI_AIT401.Sim, RIO_Hty := AI_AIT_401_HRDNSS_HTY, WRIO_Hty := W_AI_AIT_401_HRDNSS_HTY, HMI := HMI_AIT401, Pv := HMI_AIT401.Pv, Sim_PV := HMI_AIT401.Sim_PV);
   HMI_AIT401.Wifi_Enb := AIT401_FB.Wifi_Enb;
   HMI_AIT401.AHH := AIT401_FB.AHH;
   HMI_AIT401.ALL := AIT401_FB.ALL;
   HMI_AIT401.Hty := AIT401_FB.Hty;
   HMI_AIT401.AH := AIT401_FB.AH;
   HMI_AIT401.AL := AIT401_FB.AL;
   FIT401_FB : FIT_FBD(WRIO_Enb := DI_WIFI_RIO_4, Raw_RIO := AI_FIT_401_FLOW, Raw_WRIO := W_AI_FIT_401_FLOW, L_Raw_RIO := -5, H_Raw_RIO := 31208, L_Raw_WRIO := 3277, H_Raw_WRIO := 16383, HEU := 4, LEU := 0.0, SAHH := HMI_FIT401.SAHH, SAH := HMI_FIT401.SAH, SAL := HMI_FIT401.SAL, SALL := HMI_FIT401.SALL, Simulation := HMI_FIT401.Sim, RIO_Hty := AI_FIT_401_FLOW_HTY, WRIO_Hty := W_AI_FIT_401_FLOW_HTY, Totaliser_Enb := _FIT401_Tot_Enb, Rst_Totaliser := HMI_FIT401.Rst_Totaliser, HMI := HMI_FIT401, Pv := HMI_FIT401.Pv, Sim_Pv := HMI_FIT401.Sim_PV, Totaliser := HMI_FIT401.Totaliser);
   HMI_FIT401.Wifi_Enb := FIT401_FB.Wifi_Enb;
   HMI_FIT401.AHH := FIT401_FB.AHH;
   HMI_FIT401.Hty := FIT401_FB.Hty;
   HMI_FIT401.AH := FIT401_FB.AH;
   HMI_FIT401.AL := FIT401_FB.AL;
   HMI_FIT401.ALL := FIT401_FB.ALL;
END_ROUTINE

ROUTINE VALIDATE_INPUT   (* structured text *)
   (*SECOND PULSE*)
   TON.PRE	:=1000;
   TON.TimerEnable	:=1;
   TONR(TON );
   R_TRIG.InputBit :=TON.DN ;
   OSRI( R_TRIG);
   _SEC_P  := R_TRIG.OutputBit;
   TON.Reset := _SEC_P;
   
   IF  _SEC_P      THEN
   	SEC_TEST:=SEC_TEST+1;
       //_SEC_P_2 := 1;         (* we made it *)
   END_IF;
   
   IF  SEC_TEST = 60   THEN
   	_MIN_P  := 1;
   	SEC_TEST:=0;
   END_IF;
   
   
   
   
   // ESTIMATE LIT401 LEVEL
   
   //BACK CHECKING
   (* HOW TO OVER COME BACKWASH CYCLE TIME IN STATE CHECKING AND CHECK THE STATES: use MV302 status*)
   (*   *)
   (*  WHEN LIT401 LOW PUMP P301 SHOULD RUN OR MV302 SHOULD BE OPEN*)
   
   IF HMI_LIT401.AL THEN
   //TIME
   	IF HMI_P301.Status = 1  AND HMI_MV302.Status = 1 THEN
   		ATTACK :=1;
   	END_IF;
   END_IF;
   
   (*  LIT401 HIGH PUMP P301 SHOULD BE STOP  *)
   IF HMI_LIT401.AH THEN
   	//TIME
   	IF HMI_P301.Status = 2 THEN
   		ATTACK :=1;
   	END_IF;
   END_IF;
   
   
   //FORWARD CHECKING
   
   (* LIT401 LOW LOW PUMP P401 SHOULD STOP *)
   (* P401 ON FIT401 SHOULD HAVE VALUE  *)
   (* FIT401 SHOULD HAVE SOME VALUE THEN ONLY UV401 SHOULD ON  *)
   (*  FIT401 HAVE SOME VALUE THEN FIT501 ALSO HAVE SOME VALUE*)
END_ROUTINE
END_PROGRAM
